		(* split slave state and link state *)
			FOR I_X1 := 1 TO MIN(nEcSlavesRead_X1, GVL.ECAT_MAX_SLAVES_X1) DO
				(* slave state*)
				arrSlaveInfo_X1[I_X1].stState.eEcState 				:= ArrEcSlaveState_X1[I_X1].deviceState AND 16#0F;
				arrSlaveInfo_X1[I_X1].stState.bError 					:= ArrEcSlaveState_X1[I_X1].deviceState.4;
				arrSlaveInfo_X1[I_X1].stState.bInvalidVPRS 			:= ArrEcSlaveState_X1[I_X1].deviceState.5;
				(* link state *)
				arrSlaveInfo_X1[I_X1].stState.bNoCommToSlave 	:= ArrEcSlaveState_X1[I_X1].linkState.0;
				arrSlaveInfo_X1[I_X1].stState.bLinkError 				:= ArrEcSlaveState_X1[I_X1].linkState.1;
				arrSlaveInfo_X1[I_X1].stState.bMissingLink 			:= ArrEcSlaveState_X1[I_X1].linkState.2;
				arrSlaveInfo_X1[I_X1].stState.bUnexpectedLink		:= ArrEcSlaveState_X1[I_X1].linkState.3;
				arrSlaveInfo_X1[I_X1].stState.bPortA 					:= ArrEcSlaveState_X1[I_X1].linkState.4;
				arrSlaveInfo_X1[I_X1].stState.bPortB 					:= ArrEcSlaveState_X1[I_X1].linkState.5;
				arrSlaveInfo_X1[I_X1].stState.bPortC 					:= ArrEcSlaveState_X1[I_X1].linkState.6;
				arrSlaveInfo_X1[I_X1].stState.bPortD 					:= ArrEcSlaveState_X1[I_X1].linkState.7;
				(* DiagData *)
				arrSlaveInfo_X1[I_X1].bDiagData	:= ((ArrEcSlaveState_X1[I_X1].deviceState AND 16#F0) <> 0) OR
					(((ArrEcSlaveState_X1[I_X1].deviceState AND 16#0F) > 0) AND ((ArrEcSlaveState_X1[I_X1].deviceState AND 16#0F) < 8)) OR
					(ArrEcSlaveState_X1[I_X1].linkState <> 0);

				IF arrSlaveInfo_X1[I_X1].bDiagData THEN
					IF (I_X1=0) THEN
						iDiagIndex_X1[0] := 0;
					ELSE
						IF (iDiagIndex_X1[0] = 0) AND NOT arrSlaveInfo_X1[1].bDiagData THEN
							iDiagIndex_X1[0] :=  DINT_TO_UINT(I_X1);
						END_IF
					END_IF
				END_IF


				arrSlaveInfo_X1[I_X1].sName							:=	ArrEcConfSlaveInfo_X1[I_X1].sName;
				arrSlaveInfo_X1[I_X1].sType							:=	ArrEcConfSlaveInfo_X1[I_X1].sType;
				arrSlaveInfo_X1[I_X1].nECAddr						:=	ArrEcConfSlaveInfo_X1[I_X1].nAddr;

				IF arrSlaveInfo_X1[I_X1].stState.bError THEN
					sState_X1	 	:=	'ERR';
				ELSE
					sState_X1		:=	'';
				END_IF

				IF arrSlaveInfo_X1[I_X1].stState.bInvalidVPRS THEN
					sState_X1	 	:=	' VPRS INIT_ERR';
				END_IF

				IF arrSlaveInfo_X1[I_X1].stState.bNoCommToSlave THEN
					sState_X1	 	:=	CONCAT ( sState_X1, ' NO_COMM');
				END_IF

				IF arrSlaveInfo_X1[I_X1].stState.bLinkError THEN
					sState_X1	 	:=	CONCAT ( sState_X1, ' LINK_ERR');
				END_IF

				IF arrSlaveInfo_X1[I_X1].stState.bUnexpectedLink THEN
					sState_X1	 	:=	CONCAT ( sState_X1, ' UNEXP_LINK');
				END_IF

				IF arrSlaveInfo_X1[I_X1].stState.bMissingLink THEN
					sState_X1	 	:=	CONCAT ( sState_X1, ' LINK_MIS ');
				END_IF

				IF arrSlaveInfo_X1[I_X1].stState.bPortA THEN
					sState_X1	 	:=	CONCAT ( sState_X1, 'A ');
				END_IF

				IF arrSlaveInfo_X1[I_X1].stState.bPortB THEN
					sState_X1	 	:=	CONCAT ( sState_X1, 'B ');
				END_IF


				IF arrSlaveInfo_X1[I_X1].stState.bPortC THEN
					sState_X1	 	:=	CONCAT ( sState_X1, 'C ');
				END_IF

				IF arrSlaveInfo_X1[I_X1].stState.bPortD THEN
					sState_X1	 	:=	CONCAT ( sState_X1, 'D ');
				END_IF

				arrSlaveInfo_X1[I_X1].sStateString := sState_X1;
				
				CASE  arrSlaveInfo_X1[I_X1].stState.eEcState	OF 
						
						0:	arrSlaveInfo_X1[I_X1].sEcState	:= 'Úndefined';
						1:	arrSlaveInfo_X1[I_X1].sEcState	:= 'INIT';
						2:	arrSlaveInfo_X1[I_X1].sEcState	:= 'PREOP';
						3:	arrSlaveInfo_X1[I_X1].sEcState	:= 'BOOT';
						4:	arrSlaveInfo_X1[I_X1].sEcState	:= 'SAFEOP';
						8:	arrSlaveInfo_X1[I_X1].sEcState	:= 'OP';
						
				END_CASE
			END_FOR
		END_IF
	END_IF
END_IF

IF bCheckError THEN
		IF N_X1 = 0 THEN
			N_X1 :=1;
		END_IF
		IF arrSlaveInfo_X1[N_X1].sEcState <> 'OP' AND arrSlaveInfo_X1[N_X1].sEcState <> '' THEN
			CASE ErrorState_X1 OF 
				0:
					fbGetSlaveState_X1(sNetId:= sEcMasterNetId_X1,
									   nSlaveAddr:= arrSlaveInfo_X1[N_X1].nECAddr, 
									   bExecute:=TRUE,
									   tTimeout:= DEFAULT_ADS_TIMEOUT,
									   state:=EC_DEVICE_STATE_ERROR);
					ErrorState_X1 := ErrorState_X1+1;
					
				2:
					IF NOT fbGetSlaveState_X1.bBusy AND NOT fbGetSlaveState_X1.bError THEN
						fbGetSlaveState_X1(bExecute:=FALSE);
						ErrorState_X1 := ErrorState_X1+1;
					END_IF
					IF fbGetSlaveState_X1.bBusy AND fbGetSlaveState_X1.bError THEN
						ErrorState_X1 := 100;
					END_IF
				3:
					fbGetSlaveState_X1(sNetId:= sEcMasterNetId_X1,
									   nSlaveAddr:= arrSlaveInfo_X1[N_X1].nECAddr, 
									   bExecute:=TRUE,
									   tTimeout:= DEFAULT_ADS_TIMEOUT,
									   state:=EC_DEVICE_STATE_OP);
					ErrorState_X1 := ErrorState_X1+1;
				4:
					IF NOT fbGetSlaveState_X1.bBusy AND NOT fbGetSlaveState_X1.bError THEN
						fbGetSlaveState_X1(bExecute:=FALSE);
						ErrorState_X1 := ErrorState_X1+1;
					END_IF
					IF fbGetSlaveState_X1.bBusy AND fbGetSlaveState_X1.bError THEN
						ErrorState_X1 := 100;
					END_IF
				5:
					ErrorState_X1 := 0;
					N_X1 := N_X1+1;
			END_CASE;
		ELSE
			N_X1 := N_X1+1;
		END_IF;
		
		IF N_X1 = MIN(nEcSlavesRead_X1, GVL.ECAT_MAX_SLAVES_X1) THEN
			N_X1 := 1;
			bCheckError:=1;
		END_IF
END_IF;

END_PROGRAM

// ---- FB/Cylinder_Block_HOMING.TcPOU
FUNCTION_BLOCK Cylinder_Block_HOMING
VAR_INPUT
	Auto :BOOL;
	Manual :BOOL;
	HOMING_RUNNING:BOOL;
	ErrorActive :BOOL;
	ResetPB :BOOL;
	Sensor1 :BOOL;
	Sensor2 :BOOL;
	ManualPB1 :BOOL;
	ManualPB2 :BOOL;
	AutoCmd1 :BOOL;
	AutoCmd2 :BOOL;
	OperationEnable :BOOL;
	SafeHome :BOOL;
	SafeWork :BOOL;
	Pulse_1Sec :BOOL;
	BlinkingBit :BOOL;
	TimeOut1 :INT;
	TimeOut2 :INT;
	TimeOut3 :INT;
	HOMING_STRT:BOOL;
	HME_DLY:INT;
	HME_DN_NO:INT;
	HME_CYL_2:BOOL;
	HME_CYL_3:BOOL;
END_VAR
VAR_OUTPUT
	Solenoid1 :BOOL;
	Solenoid2 :BOOL;
	AlarmSensor1 :BOOL;
	AlarmSensor2 :BOOL;
	AlarmSolenoid1 :BOOL;
	AlarmSolenoid2 :BOOL;
	AllSignal :BOOL;
	AlarmPresent :BOOL;
	Position1 :BOOL;
	Position2 :BOOL;
	HomeSensorBlink :BOOL;
	WorkSensorBlink :BOOL;
END_VAR
VAR_IN_OUT
	Status :INT;
	HMENG_RESULT: INT;
END_VAR
VAR
	Timer1 :INT;
	Timer2 :INT;
	Timer3 :INT;
	HomingCmd1:BOOL;
	HomePositionErr_1SecPls :Tc2_Standard.R_TRIG;
	WorkPositionErr_1SecPls :Tc2_Standard.R_TRIG;
	BothSensorErr_1SecPls :Tc2_Standard.R_TRIG;
	Temp4 :BOOL;
	AFT_CYL_HME: TON;
END_VAR

Status:=0;
//Cylinder Moving to Home Position by Manual

IF ManualPB1 THEN
	IF NOT Manual THEN Status :=1; 
	ELSIF ManualPB2 THEN Status :=2; 
	ELSIF AllSignal THEN Status :=3;
	ELSIF NOT OperationEnable THEN Status :=9; 
	ELSIF Status =0 AND SafeHome THEN
		Solenoid1 :=1;
		Solenoid2 :=0;
	END_IF 
END_IF


//Cylinder Moving to Work Position by Manual

IF ManualPB2 THEN
	IF NOT Manual THEN Status :=1; 
	ELSIF ManualPB1 THEN Status :=2; 
	ELSIF AllSignal THEN Status :=3;
	ELSIF NOT OperationEnable THEN Status :=9; 
	ELSIF Status =0 AND SafeWork THEN
		Solenoid2 :=1;
		Solenoid1 :=0;
	END_IF 
END_IF


//Cylinder Moving to Home Position by Auto

IF AutoCmd1 THEN
	IF NOT Auto THEN Status :=5; 
	ELSIF AutoCmd2 THEN Status :=6;
	ELSIF ErrorActive THEN Status :=4; 
	ELSIF AllSignal THEN Status :=3;
	ELSIF NOT OperationEnable THEN Status :=9;
	ELSIF Status =0 AND SafeHome THEN
		Solenoid1 :=1;
		Solenoid2 :=0;
	END_IF 
END_IF

//Cylinder Moving to Work Position by Auto

IF AutoCmd2 THEN
	IF NOT Auto THEN Status :=5; 
	ELSIF AutoCmd1 THEN Status :=6;
	ELSIF ErrorActive THEN Status :=4; 
	ELSIF AllSignal THEN Status :=3;
	ELSIF NOT OperationEnable THEN Status :=9;
	ELSIF Status =0 AND SafeWork THEN
		Solenoid2 :=1;
		Solenoid1 :=0;
	END_IF 
END_IF


//Cylinder Moving to Home Position - Homing Cmd ON

IF HomingCmd1 THEN 
	IF AllSignal THEN Status :=3;
	ELSIF NOT OperationEnable THEN Status :=9; 
	ELSIF Status =0 AND SafeHome THEN
		Solenoid1 :=1;
		Solenoid2 :=0;
	END_IF 
END_IF


// While Cylinder Moving Blinking IF Position Reached then Steady Indication

HomeSensorBlink := (Solenoid1 AND NOT Sensor1 AND BlinkingBit) OR Sensor1;
WorkSensorBlink := (Solenoid2 AND NOT Sensor2 AND BlinkingBit) OR Sensor2;


// Position 1 Reached - Cylinder Timer OFF

IF NOT Solenoid1 THEN Timer1 :=0; END_IF


//Timer1 is for Monitoring Cylinder Home Position Time
HomePositionErr_1SecPls(CLK := Pulse_1Sec);

IF Solenoid1 AND NOT Sensor1 AND HomePositionErr_1SecPls.Q THEN 
Timer1 := Timer1 + 1;
ELSE
Timer1	:= 0;	
END_IF


//Generate Alarm for Home Position Sensor & Valve

IF Timer1 >= TimeOut1 AND NOT Sensor1 AND NOT Sensor2 THEN AlarmSensor1 :=1; END_IF
IF Timer1 >= TimeOut1 AND NOT Sensor1 AND Sensor2 THEN AlarmSolenoid1 :=1; END_IF


// Position 2 Reached - Cylinder Timer OFF

IF NOT Solenoid2 THEN Timer2 :=0; END_IF


//Timer2 is for Monitoring Cylinder Work Position Time
WorkPositionErr_1SecPls(CLK := Pulse_1Sec);

IF Solenoid2 AND NOT Sensor2 AND WorkPositionErr_1SecPls.Q THEN 
	Timer2 := Timer2 + 1;
ELSE
	Timer2	:=0;
END_IF


//Generate Alarm for Work Position Sensor & Valve

IF Timer2 >= TimeOut2 AND NOT Sensor2 AND NOT Sensor1 THEN AlarmSensor2 :=1; END_IF
IF Timer2 >= TimeOut2 AND NOT Sensor2 AND Sensor1 THEN AlarmSolenoid2 :=1; END_IF


//Move "0" to Timer3 If anyone Sensor is not Sensing

IF NOT Sensor1 AND NOT Sensor2 THEN Timer3 :=0; END_IF


//Timer3 is for Monitoring Both Sensor ON Error
BothSensorErr_1SecPls (CLK := Pulse_1Sec);

 IF Sensor1 AND Sensor2 AND BothSensorErr_1SecPls.Q THEN
	 Timer3 := Timer3 + 1;
 END_IF
 
 
 //Generate Alarm for Both Sensor ON Error
 
 IF Timer3 >= TimeOut3 THEN AllSignal :=1; END_IF
 
 
 //Reset the Valve when Operation Enable not Present
 
 IF NOT OperationEnable THEN
	 Solenoid1 :=0;
	 Solenoid2 :=0;
 END_IF

 
//Position 1 is Cylinder Home Position || Position 2 is Cylinder Work Position

Position1 := NOT AllSignal AND Sensor1 AND NOT Sensor2;
Position2 := NOT AllSignal AND Sensor2 AND NOT Sensor1; 

// HOMING LOGIC

IF HOMING_RUNNING AND HOMING_STRT AND NOT ErrorActive THEN
	HomingCmd1				:= TRUE;
ELSE
	HomingCmd1				:= FALSE;
END_IF

AFT_CYL_HME(IN:= (HomingCmd1 AND HME_CYL_2 AND HME_CYL_3 AND Sensor1 AND NOT ErrorActive), PT:=INT_TO_TIME(HME_DLY) , Q=> , ET=> );
IF AFT_CYL_HME.Q THEN
	HMENG_RESULT:=HME_DN_NO;
END_IF

// ALARM RESET

IF ResetPB THEN
	
AlarmSensor1 								:= FALSE;
AlarmSensor2            					:= FALSE;
AlarmSolenoid1          					:= FALSE;
AlarmSolenoid2          					:= FALSE;
AllSignal               					:= FALSE;

END_IF


IF AlarmSensor1 OR AlarmSensor2 OR AlarmSolenoid1 OR AlarmSolenoid2 OR AllSignal THEN
		AlarmPresent						:= TRUE;
ELSE
		AlarmPresent						:= FALSE;
END_IF

END_FUNCTION_BLOCK

// ---- FB/Axis/FB_Axis_FESTO.TcPOU
FUNCTION_BLOCK FB_Axis_FESTO
VAR_INPUT
	bAxis1_Ref_Switch 	 : BOOL;//HW-IN
	bInit 				 : BOOL;
	bErrorReset			 : BOOL;//FP Reset Axis Error
	bEnable 			 : BOOL;//Power on
	bMoveVelocity 		 : BOOL;
	bHalt				 : BOOL;//Stop Absolute or Relative movement
	bManualMode			 : BOOL;
	bmove_home			 : BOOL;
	fHomePos 			 : LREAL := 0.0;
	fOverride 			 : LREAL ;//:= 100.0;
	fTargetPosition 	 : LREAL ;//:=  10.0;
	fTargetVelocity 	 : LREAL ; //:= 100.0;
	fAcc				 : LREAL; //:= 100.0;
	fDec				 : LREAL; //:= 100.0;
	Servo_High_Limit	 : LREAL;
	Servo_Low_Limit	 	 : LREAL;
	WARNING_LIMIT		 : LREAL;
	Safe_move_Conditions : BOOL;
	LIMIT_BYPASS		 : BOOL := TRUE;
	TORQUE_APPLIED: LREAL;
END_VAR
VAR_IN_OUT
	Axis 				: AXIS_REF;
	bHome 				: BOOL;
	bSetPosition		: BOOL;//Set Position to HomePos
	bMoveAbsolute 		: BOOL;
	bMoveRelative 		: BOOL;
	bMoveTorque			: BOOL;
    stManualModeAxis  	: stManualModeAxis;
														(*bmove_home			: BOOL;*)
END_VAR

VAR_OUTPUT
	sAxisState			: STRING := '';
	bAxis_ready			: BOOL := 0;
	bAxisInPosition		: BOOL := 0;//In Position or In Target Velocity
	bAxisError			: BOOL := 0;
	bAxisEnabled 		: BOOL := 0;//Power ON
	bAxisHomed			: BOOL := 0;
	bSetPositionDone	: BOOL := 0;
	bHaltDone			: BOOL := 0;
	bSTOPDone			: BOOL := 0;
	bHomeDone			: BOOL := 0;
	bDone				: BOOL := 0;//bMoveAbsolute + bMoveRelative
	bTorqueReached		: BOOL := 0;
	bsafe_to_move		: BOOL;
	baxis_in_home_pos	: BOOL;
	bABS_Pos_done		: BOOL;
	Actual_position		: LREAL;
	Actual_velocity		: LREAL;
	Actual_Torque		: LREAL;
    SERVO_LIMIT_WARNING	: BOOL;	
	
END_VAR
VAR
	temp : LREAL;
	fbAxisReset					: MC_Reset;
	fbAxisPower					: MC_Power;
	fbAxisStop        			: MC_Stop;
	fbAxisHalt        			: MC_Halt;
(*	fbAxisHome					: MC_Home;*)
	fbAxisHome					: Festo_MC_Home;
	fbAxisSetPosition 			: MC_SetPosition;
	fbAxisJog 					: MC_Jog;
	fbAxisMoveAbsolute			: MC_MoveAbsolute;
	fbAxisMoveRelative 			: MC_MoveRelative;
	fbAxisMoveVelocity			: MC_MoveVelocity;
	fbAxisTorqueControl			: MC_TorqueControl;
//Brake Controll
	fbEcCoeSdoRead				: FB_EcCoeSdoRead;
	fbEcCoeSdoWrite				: FB_EcCoeSdoWrite;
	mcReadDriveAddress 			: MC_ReadDriveAddress;
    vendorId   					: BOOL;//Struct HMI Brake open
	bBrakeStateOld 				: BOOL;

//Status Information
	bAxisIsEnabled 				: BOOL;
	bAxisIsHomed 				: BOOL;
	bAxisInError 				: BOOL;
	fActualTorque 				: LREAL;	

//Allgemein
	iSchritt 					: ENUM_Axis;
	bHMFPErrorReset 			: BOOL;
	bFPErrorReset 				: BOOL;
	
	bAxisResetExecute			: BOOL;
	bAxisPowerExecute			: BOOL;
	bAxisStopExecute        	: BOOL;
	bAxisHaltExecute        	: BOOL;
	bAxisHomeExecute			: BOOL;
	bAxisSetPositionExecute 	: BOOL;
	bAxisMoveAbsoluteExecute	: BOOL;
	bAxisMoveRelativeExecute 	: BOOL;
	bAxisMoveVelocityExecute	: BOOL;
	bAxisJogExecutePos 			: BOOL;
	bAxisJogExecuteNeg 			: BOOL;
	bAxisMoveTorqueExecute		: BOOL;
	fHMTargetPosition			: LREAL;
	fHMTargetVelocity			: LREAL;
	
	bFPManualReset				: BOOL;
	bHMFPManualReset			: BOOL;
	
	homeMode					: MC_HomingMode;
	FB_SoEReset					: FB_SoEReset;
	bHardwareReset				: BOOL;

	st_Trq_options 				: St_TorqueControlOptions;
	//temp						: BOOL;
	moving_home					: INT;
	bABS_done					: BOOL;
	busy: BOOL;
	act: BOOL;
	id: UDINT;
	AXIS_REF_TEMP: BOOL;
	
	LEG_LIMIT: BOOL;
	POS_LIMIT: BOOL;
	AUTO_TARGET_POSITION: LREAL;
	MANUAL_TARGET_POSITION: LREAL;
	ABS_BUSY: R_TRIG;
END_VAR
VAR_TEMP
 	//tmpVelocityDirection		: MC_Direction;
	tmpStManualModeAxis	  		: stManualModeAxis;
	btmpFPBrake					: BOOL;
//	tmpVelocityDirection        : MC_Direction;
END_VAR


//Init
bHaltDone := FALSE;
bSTOPDone := FALSE;

//Read Axis Status	
	bAxisIsEnabled := axis.NcToPlc.StateDWord.0;
	bAxisIsHomed := axis.NcToPlc.StateDWord.1 OR NOT AXIS_REF_TEMP;
	bAxisInError := axis.NcToPlc.StateDWord.31;
	fActualTorque := axis.NcToPlc.ActTorque;
    Axis.ReadStatus(); // PHU: fill its own status bits.
//FP Error Reset
	bFPErrorReset := bErrorReset (*AND NOT bHMFPErrorReset*);
	bHMFPErrorReset := bErrorReset;
	
	bFPManualReset:= stManualModeAxis.reset AND NOT bHMFPManualReset;
	bHMFPManualReset:= stManualModeAxis.reset;
	
// Manual Mode
IF bManualMode THEN
	
	stManualModeAxis.stationModeAutoManual:= FALSE;	
	IF 	stManualModeAxis.jogPos THEN
		tmpStManualModeAxis.jogPos := TRUE;
	ELSE
		tmpStManualModeAxis.jogPos := FALSE;		
	END_IF
	IF 	stManualModeAxis.jogNeg THEN
		tmpStManualModeAxis.jogNeg := TRUE;
	ELSE
		tmpStManualModeAxis.jogNeg := FALSE;		
	END_IF
		
ELSE
	stManualModeAxis.jogPos := FALSE;
	stManualModeAxis.jogNeg := FALSE;
	stManualModeAxis.reset := FALSE;
	StManualModeAxis.openBrake:= FALSE;
	stManualModeAxis.homing:= FALSE;
	stManualModeAxis.moveAbsolute:= FALSE;
	stManualModeAxis.moveRelative:= FALSE;
	stManualModeAxis.moveVelocity:= FALSE;
	
	tmpStManualModeAxis.jogPos := FALSE;		
	tmpStManualModeAxis.jogNeg := FALSE;	
	
	
	
	stManualModeAxis.stationModeAutoManual:= TRUE;

END_IF


//###################################################################################
//###################################################################################	
	
//###################################################################################
//###################################################################################

	CASE iSchritt OF 
		
	ENUM_Axis.Init 			://init all MC
								bAxisResetExecute				:= FALSE;
								bAxisPowerExecute				:= FALSE;
								bAxisStopExecute        		:= FALSE;
								bAxisHaltExecute        		:= FALSE;
								bAxisHomeExecute				:= FALSE;
								bAxisSetPositionExecute 		:= FALSE;
								bAxisJogExecutePos 				:= FALSE;
								bAxisJogExecuteNeg 				:= FALSE;
								bAxisMoveAbsoluteExecute		:= FALSE;
								bAxisMoveRelativeExecute 		:= FALSE;
								bAxisMoveVelocityExecute		:= FALSE;
								
								iSchritt := ENUM_Axis.PowerOFF;
								

	ENUM_Axis.PowerOFF		: 	//Power off
								bAxisPowerExecute		:= FALSE;
								IF bInit THEN
									iSchritt := ENUM_Axis.Init;
								ELSIF bAxisInError THEN
									iSchritt := ENUM_Axis.Error;
								ELSIF bEnable THEN
									iSchritt := ENUM_Axis.PowerON;
								END_IF
								
	ENUM_Axis.Error			:	//Error
								bAxisPowerExecute			  := FALSE;
								bMoveAbsolute				  := FALSE;
								bMoveRelative			   	  := FALSE;
								stManualModeAxis.moveAbsolute := FALSE;
								stManualModeAxis.moveRelative := FALSE;
								IF bInit THEN
									iSchritt := ENUM_Axis.Init;
								ELSIF bFPErrorReset OR bFPManualReset THEN
									iSchritt := ENUM_Axis.Reset;
								END_IF
	ENUM_Axis.Reset			: //Error Reset
								IF NOT fbAxisReset.Busy THEN
									bAxisResetExecute 		:= TRUE;
									bHardwareReset			:= axis.NcToPlc.StateDWord.28;
								END_IF;
								IF bInit THEN
									bAxisResetExecute 		:= FALSE;
									iSchritt := ENUM_Axis.Init;
								ELSIF fbAxisReset.Error (*OR bAxisInError *)THEN
									bAxisResetExecute 	:= FALSE;
									iSchritt := ENUM_Axis.Error;
								ELSIF fbAxisReset.Done AND NOT bAxisInError THEN
									bAxisResetExecute 	:= FALSE;
									IF  bAxisInError THEN
										iSchritt := ENUM_Axis.Error;
									ELSE
										iSchritt := ENUM_Axis.PowerOFF;
									END_IF
								END_IF

	ENUM_Axis.PowerON		:	//Enable - Power on
								bAxisPowerExecute := TRUE;
								IF bInit THEN
									bAxisPowerExecute 	:= FALSE;
									iSchritt := ENUM_Axis.Init;
								ELSIF NOT benable THEN
									iSchritt:= enum_axis.PowerOFF;
								ELSIF fbAxisPower.Error OR bAxisInError THEN
									bAxisPowerExecute 	:= FALSE;
									iSchritt := ENUM_Axis.Error;
								ELSIF fbAxisPower.Status THEN
									iSchritt := ENUM_Axis.Ready;
								END_IF
	ENUM_Axis.Stop			://Axis Stop
								bAxisStopExecute := TRUE;
								IF bInit THEN
									bAxisStopExecute 	:= FALSE;
									iSchritt := ENUM_Axis.Init;
								ELSIF NOT benable THEN
									bAxisStopExecute 	:= FALSE;
									iSchritt:= enum_axis.PowerOFF;	
								ELSIF fbAxisStop.Error OR bAxisInError THEN
									bAxisStopExecute := FALSE;
									iSchritt := ENUM_Axis.Error;
								ELSIF fbAxisStop.Done THEN
									bSTOPDone	:= TRUE;
									bAxisStopExecute 	:= FALSE;
									iSchritt := ENUM_Axis.PowerOFF;
								END_IF
	ENUM_Axis.Halt			://Axis Halt
								bAxisHaltExecute := TRUE;
								IF bInit THEN
									bAxisHaltExecute 	:= FALSE;
									iSchritt := ENUM_Axis.Init;
								ELSIF NOT benable THEN
									bAxisHaltExecute 	:= FALSE;
									iSchritt:= enum_axis.PowerOFF;	
								ELSIF bAxisInError THEN
									bAxisHaltExecute := FALSE;
									iSchritt := ENUM_Axis.Error;
								ELSIF fbAxisHalt.Error (*OR bAxisInError *)THEN
									bAxisHaltExecute := FALSE;
									iSchritt := ENUM_Axis.Stop;
								ELSIF fbAxisHalt.Done THEN
									bHaltDone := TRUE;
									bAxisHaltExecute := FALSE;
									iSchritt := ENUM_Axis.Ready;
								END_IF
	ENUM_Axis.Ready			: 	//Wait for command
								bAxisInPosition := FALSE;
								//bHomeDone := FALSE;
								bSetPositionDone := FALSE;
								IF bInit THEN
									iSchritt := ENUM_Axis.Init;
								ELSIF NOT benable THEN
									iSchritt:= enum_axis.PowerOFF;		
								ELSIF bAxisInError THEN
									iSchritt := ENUM_Axis.Error;
								ELSE
									IF bHome OR stManualModeAxis.homing THEN
										iSchritt := ENUM_Axis.Homing;
									ELSIF bSetPosition THEN
											iSchritt := ENUM_Axis.SetPosition;
									ELSIF bAxisIsHomed THEN
										IF tmpStManualModeAxis.jogPos THEN
											iSchritt := ENUM_Axis.JogPos;
										ELSIF tmpStManualModeAxis.jogNeg THEN
											iSchritt := ENUM_Axis.JogNeg;
										ELSIF bMoveAbsolute OR stManualModeAxis.moveAbsolute  THEN
											iSchritt := ENUM_Axis.MoveAbsolute;
										ELSIF bMoveRelative OR stManualModeAxis.moveRelative THEN
											iSchritt := ENUM_Axis.MoveRelative;
										ELSIF bMoveVelocity OR stManualModeAxis.moveVelocity THEN
											iSchritt := ENUM_Axis.MoveVelocity;
										ELSIF bMoveTorque OR stManualModeAxis.moveTorque THEN
											iSchritt := ENUM_Axis.MoveTorque;
										END_IF
									END_IF	
								END_IF							
	ENUM_Axis.Homing		://Homing
								IF NOT fbAxisHome.Busy THEN
									bAxisHomeExecute := TRUE;
									bHomeDone		:= FALSE;
								END_IF;
								IF bInit THEN
									bAxisHomeExecute 	:= FALSE;
									iSchritt := ENUM_Axis.Init;
								ELSIF NOT benable THEN
									bAxisHomeExecute:= FALSE;
									iSchritt:= enum_axis.PowerOFF;	
								ELSIF fbAxisHome.Error OR bAxisInError THEN
									bAxisHomeExecute:= FALSE;
									iSchritt := ENUM_Axis.Error;
								ELSIF fbAxisHome.Done THEN
									bHomeDone	:= TRUE;
									bHome := FALSE;
									stManualModeAxis.homing:= FALSE;
									bAxisHomeExecute:= FALSE;
									iSchritt := ENUM_Axis.Ready;
								END_IF
	
	ENUM_Axis.SetPosition	://Enable - Power on
								IF NOT fbAxisSetPosition.Busy THEN
									bAxisSetPositionExecute := TRUE;
								END_IF;
								IF bInit THEN
									bAxisSetPositionExecute 	:= FALSE;
									iSchritt := ENUM_Axis.Init;
								ELSIF NOT benable THEN
									bAxisSetPositionExecute 	:= FALSE;
									iSchritt:= enum_axis.PowerOFF;		
								ELSIF fbAxisSetPosition.Error OR bAxisInError THEN
									bAxisSetPositionExecute 	:= FALSE;
									iSchritt := ENUM_Axis.Error;
								ELSIF fbAxisSetPosition.Done THEN
									bAxisSetPositionExecute 	:= FALSE;
									bSetPositionDone := TRUE;
									bSetPosition := FALSE;
									iSchritt := ENUM_Axis.Ready;
								END_IF

	ENUM_Axis.JogPos		://Jog positive direction
								IF NOT fbAxisJog.Busy THEN
									bAxisJogExecutePos 		:= TRUE;
								END_IF;
								
								IF bInit THEN
									bAxisJogExecutePos 	:= FALSE;
									iSchritt := ENUM_Axis.Init;
								ELSIF NOT benable THEN
									bAxisJogExecutePos 	:= FALSE;
									iSchritt:= enum_axis.PowerOFF;			
								ELSIF fbAxisJog.Error OR bAxisInError THEN
									bAxisJogExecutePos 		:= FALSE;
									iSchritt := ENUM_Axis.Error;
								ELSIF NOT tmpStManualModeAxis.jogPos THEN
									bAxisJogExecutePos 		:= FALSE;
									iSchritt := ENUM_Axis.Ready;
								END_IF;
	ENUM_Axis.JogNeg		://Jog negative direction
								IF NOT fbAxisJog.Busy THEN
									bAxisJogExecuteNeg 		:= TRUE;
								END_IF;
								
								IF bInit THEN
									bAxisJogExecuteNeg 	:= FALSE;
									iSchritt := ENUM_Axis.Init;
								ELSIF NOT benable THEN
									bAxisJogExecuteNeg 	:= FALSE;
									iSchritt:= enum_axis.PowerOFF;		
								ELSIF fbAxisJog.Error OR bAxisInError THEN
									bAxisJogExecuteNeg 		:= FALSE;
									iSchritt := ENUM_Axis.Error;
								ELSIF NOT tmpStManualModeAxis.jogNeg THEN
									bAxisJogExecuteNeg 		:= FALSE;
									iSchritt := ENUM_Axis.Ready;
								END_IF;
	ENUM_Axis.MoveAbsolute	://MoveAbsolute
								IF NOT fbAxisMoveAbsolute.Busy THEN
									bAxisMoveAbsoluteExecute := TRUE;
								END_IF;
								IF bInit THEN
									bAxisMoveAbsoluteExecute 	:= FALSE;
									iSchritt := ENUM_Axis.Init;
								ELSIF NOT benable THEN
									bAxisMoveAbsoluteExecute 	:= FALSE;
									iSchritt:= enum_axis.PowerOFF;		
								ELSIF fbAxisMoveAbsolute.Error OR bAxisInError THEN
									bAxisMoveAbsoluteExecute :=FALSE;
									iSchritt := ENUM_Axis.Error;
								ELSIF bHalt THEN
									bMoveAbsolute :=FALSE;
									stManualModeAxis.moveAbsolute:= FALSE;
									bAxisMoveAbsoluteExecute :=FALSE;
									iSchritt := ENUM_Axis.Halt;
								ELSIF fbAxisMoveAbsolute.Done THEN
								//ELSIF fbAxisMoveAbsolute.Done AND NOT bMoveAbsolute THEN
									bMoveAbsolute :=FALSE;
									stManualModeAxis.moveAbsolute:= FALSE;
									bAxisInPosition := TRUE;
									bAxisMoveAbsoluteExecute :=FALSE;
									iSchritt := ENUM_Axis.Ready;
								END_IF;
	ENUM_Axis.MoveRelative	://MoveRelative
								IF NOT fbAxisMoveRelative.Busy THEN
									bAxisMoveRelativeExecute := TRUE;
								END_IF;
								IF bInit THEN
									bAxisMoveRelativeExecute 	:= FALSE;
									iSchritt := ENUM_Axis.Init;
								ELSIF NOT benable THEN
									bAxisMoveRelativeExecute 	:= FALSE;
									iSchritt:= enum_axis.PowerOFF;		
								ELSIF fbAxisMoveRelative.Error OR bAxisInError THEN
									bAxisMoveRelativeExecute :=FALSE;
									iSchritt := ENUM_Axis.Error;
								ELSIF bHalt THEN
									bMoveRelative :=FALSE;
									stManualModeAxis.moveRelative:= FALSE;
									bAxisMoveRelativeExecute :=FALSE;
									iSchritt := ENUM_Axis.Halt;
								ELSIF fbAxisMoveRelative.Done THEN
									bMoveRelative :=FALSE;
									stManualModeAxis.moveRelative:= FALSE;
									bAxisInPosition := TRUE;
									bAxisMoveRelativeExecute :=FALSE;
									iSchritt := ENUM_Axis.Ready;
								END_IF;
	ENUM_Axis.MoveVelocity	://MoveVelocity
								IF NOT fbAxisMoveVelocity.Busy THEN
									bAxisMoveVelocityExecute := TRUE;				
								END_IF;
								
								bAxisInPosition := fbAxisMoveVelocity.InVelocity;
								IF bInit THEN
									bAxisMoveVelocityExecute 	:= FALSE;
									bAxisInPosition := FALSE;
									iSchritt := ENUM_Axis.Init;
								ELSIF NOT benable THEN
									bAxisMoveVelocityExecute 	:= FALSE;
									iSchritt:= enum_axis.PowerOFF;		
								ELSIF fbAxisMoveVelocity.Error OR bAxisInError THEN
									bAxisInPosition := FALSE;
									bAxisMoveVelocityExecute :=FALSE;
									iSchritt := ENUM_Axis.Error;
								ELSIF NOT bMoveVelocity AND NOT stManualModeAxis.moveVelocity THEN
									bAxisInPosition := FALSE;
									bAxisMoveVelocityExecute :=FALSE;
									iSchritt := ENUM_Axis.Halt;
								END_IF;
								
	ENUM_Axis.MoveTorque  :		IF NOT fbAxisTorqueControl.Busy THEN
									bAxisMoveTorqueExecute := TRUE;
								END_IF;
								IF bInit THEN
									bAxisMoveTorqueExecute 	:= FALSE;
									iSchritt := ENUM_Axis.Init;
								ELSIF NOT benable THEN
									bAxisMoveTorqueExecute 	:= FALSE;
									iSchritt:= enum_axis.PowerOFF;		
								ELSIF fbAxisTorqueControl.Error OR bAxisInError THEN
									bAxisMoveTorqueExecute :=FALSE;
									iSchritt := ENUM_Axis.Error;
								ELSIF bHalt THEN
									bMoveTorque	 :=FALSE;
									stManualModeAxis.moveTorque:= FALSE;
									bAxisMoveTorqueExecute :=FALSE;
									iSchritt := ENUM_Axis.Halt;
								ELSIF fbAxisTorqueControl.InTorque THEN
								//ELSIF fbAxisMoveAbsolute.Done AND NOT bMoveAbsolute THEN
									bMoveTorque :=FALSE;
									stManualModeAxis.moveTorque:= FALSE;
									bAxisInPosition := TRUE;
									bAxisMoveTorqueExecute :=FALSE;
									iSchritt := ENUM_Axis.Ready;
								END_IF;					

	END_CASE;
	
	
	stManualModeAxis.axisState:= TO_STRING(iSchritt);
//###################################################################################
//###################################################################################
//###################################################################################
//###################################################################################



fbAxisReset(
	Axis:= Axis, 
	Execute:= bAxisResetExecute , 
	Done=> , 
	Busy=> , 
	Error=> , 
	ErrorID=> );
	
fbAxisPower(
	Axis:= Axis, 
	Enable:= bAxisPowerExecute, 
	Enable_Positive:= bAxisPowerExecute, 
	Enable_Negative:= bAxisPowerExecute, 
	Override:= fOverride, 
	//BufferMode:= , 
	//Options:= , 
	Status=> , 
	Busy=> , 
	Active=> , 
	Error=> , 
	ErrorID=> );
	
fbAxisStop(
	Axis:= Axis, 
	Execute:= bAxisStopExecute, 
	Deceleration:= fDec, 
	Jerk:= 0, 
	//Options:= , 
	Done=> , 
	Busy=> , 
	Active=> , 
	CommandAborted=> , 
	Error=> , 
	ErrorID=> );
	
fbAxisHalt(
	Axis:= Axis, 
	Execute:= bAxisHaltExecute, 
	Deceleration:= fDec, 
	Jerk:= 0, 
	//BufferMode:= , 
	//Options:= , 
	Done=> , 
	Busy=> , 
	Active=>, 
	CommandAborted=> , 
	Error=> , 
	ErrorID=> );

//Homingmode
IF bAxisHomeExecute THEN
	//HomeMode := MC_DefaultHoming;
	HomeMode := MC_Direct;
ELSIF bAxisSetPositionExecute THEN
	//HomeMode := MC_ForceCalibration;
		HomeMode := MC_Direct;
END_IF;


IF bManualMode THEN
	fHMTargetPosition:= MANUAL_TARGET_POSITION;
	fHMTargetVelocity:= stManualModeAxis.targetVelocity;
ELSE
	fHMTargetPosition:=AUTO_TARGET_POSITION;
	fHMTargetVelocity:=fTargetVelocity;
END_IF


(*fbAxisHome(
	Axis:= Axis, 
	Execute:= bAxisHomeExecute OR bAxisSetPositionExecute , 
	Position:= fHomePos, 
	HomingMode:= HomeMode, //MC_DefaultHoming,//, MC_Block
	//BufferMode:= , 
	Options:= , 
	bCalibrationCam:= bAxis1_Ref_Switch, 
	Done=> , 
	Busy=> , 
	Active=> , 
	CommandAborted=> , 
	Error=> , 
	ErrorID=> );*)

fbAxisHome(
	Axis:= Axis, 
	Execute:= bAxisHomeExecute OR bAxisSetPositionExecute , 
	TimeoutTimeHomingRun:= T#1M, 
	Done=> , 
	Busy=> , 
	Error=> , 
	ErrorID=> , 
	ErrorString=> );	
	
fbAxisSetPosition(
	Axis:= Axis, 
	Execute:= bAxisSetPositionExecute, 
	Position:= fHomePos, 
	Mode:= FALSE, (* RELATIVE=True, ABSOLUTE=False (Default) *)
	//Options:= , 
	Done=> , 
	Busy=> , 
	Error=> , 
	ErrorID=> );

fbAxisJog(
	Axis:= Axis, 
	JogForward:=bAxisJogExecutePos AND (POS_LIMIT OR LIMIT_BYPASS),
	JogBackwards:= bAxisJogExecuteNeg AND (LEG_LIMIT OR LIMIT_BYPASS),
	//Mode:= MC_JOGMODE_STANDARD_SLOW, //MC_JOGMODE_STANDARD_SLOW, //MC_JOGMODE_STANDARD_FAST, //MC_JOGMODE_CONTINOUS, //MC_JOGMODE_INCHING, //MC_JOGMODE_INCHING_MODULO
	//Position:= 0, 
	Velocity:= stManualModeAxis.targetVelocity, 
	Acceleration:= fAcc, 
	Deceleration:= fDec, 
	Jerk:= 0, 
	Done=> , 
	Busy=> , 
	Active=> , 
	CommandAborted=> , 
	Error=> , 
	ErrorID=> );
	
fbAxisMoveAbsolute(
	Axis:= Axis, 
	Execute:= bAxisMoveAbsoluteExecute, 
	Position:= fHMTargetPosition,
	Velocity:= ABS(fHMTargetVelocity),
	Acceleration:= fAcc,
	Deceleration:= fDec,
	Jerk:= 0, 
	//BufferMode:= , 
	//Options:= , 
	Done=> , 
	Busy=> , 
	Active=> (bABS_done) , 
	CommandAborted=> , 
	Error=> , 
	ErrorID=> );

	ABS_BUSY(CLK:= bABS_done, Q=> );
	IF ABS_BUSY.Q THEN
	bABS_Pos_done			:= FALSE;	
	END_IF
	IF fbAxisMoveAbsolute.Done THEN
	bABS_Pos_done			:= TRUE;	
	END_IF
	
	
	
fbAxisMoveRelative(
	Axis:= Axis, 
	Execute:= bAxisMoveRelativeExecute, 
	Distance:= fHMTargetPosition, 
	Velocity:= fHMTargetVelocity, 
	Acceleration:= fAcc, 
	Deceleration:= fDec, 
	Jerk:= 0, 
	//BufferMode:= , 
	//Options:= , 
	Done=> , 
	Busy=> , 
	Active=> , 
	CommandAborted=> , 
	Error=> , 
	ErrorID=> );

IF 	fHMTargetVelocity >= 0 THEN  // fHMTargetVelocity>= 0
	fbAxisMoveVelocity.Direction:= MC_Positive_Direction;
ELSE
	fbAxisMoveVelocity.Direction:= MC_Negative_Direction;
END_IF
	
fbAxisMoveVelocity(
	Axis:= Axis, 
	Execute:= bAxisMoveVelocityExecute, 
	Velocity:=ABS(fHMTargetVelocity), 
	Acceleration:= fAcc, 
	Deceleration:= fDec, 
	Jerk:= 0, 
	Direction:= ,//MC_Negative_Direction ,//OR MC_Positive_Direction, //tmpVelocityDirection,//MC_Undefined_Direction, //MC_Shortest_Way, //MC_Positive_Direction, //MC_Negative_Direction,
	//BufferMode:= , 
	//Options:= , 
	InVelocity=> , 
	Busy=> , 
	Active=> , 
	CommandAborted=> , 
	Error=> , 
	ErrorID=> );
	
//Brake controll
vendorId	:= StManualModeAxis.openBrake;	
btmpFPBrake :=  bBrakeStateOld <> vendorId;
bBrakeStateOld := vendorId;

mcReadDriveAddress(
	Axis:= Axis, 
	Execute:= btmpFPBrake, 
	Done=> , 
	Busy=> , 
	Error=> , 
	ErrorID=> , 
	DriveAddress=> Axis.DriveAddress);

	st_Trq_options.EnableManualTorqueStartValue :=TRUE;
	st_Trq_options.ManualTorqueStartValue:= 0.5;
	bTorqueReached:=fbAxisTorqueControl.InTorque;
	
fbAxisTorqueControl	(
	Axis:= Axis , 
	Execute:=bAxisMoveTorqueExecute , 
	Relative:= , 
	Torque:= TORQUE_APPLIED, 
	TorqueRamp:= 50, 
	VelocityLimitHigh:= 500, 
	VelocityLimitLow:= -500, 
	BufferMode:= , 
	Options:= ,//st_Trq_options , 
	InTorque=> , 
	Busy=> busy, 
	Active=> , 
	CommandAborted=> , 
	Error=> act, 
	ErrorId=> id );

//	fbEcCoeSdoRead(
//	sNetId:= Axis.DriveAddress.NetID,
//	nSlaveAddr:= Axis.DriveAddress.SlaveAddress,
//	nSubIndex:= 16#1, 
//	nIndex:= 16#8012, 
//	pDstBuf:= ADR(bBrakeStateOld), 
//	cbBufLen:= SIZEOF(bBrakeStateOld), 
//	bExecute:= mcReadDriveAddress.done, 
//	tTimeout:= , 
//	bBusy=> , 
//	bError=> , 
//	nErrId=> , 
//	cbRead=> );

fbEcCoeSdoWrite(
	sNetId:= Axis.DriveAddress.NetID,
	nSlaveAddr:= Axis.DriveAddress.SlaveAddress, 
	nSubIndex:= 16#1, 
	nIndex:= 16#8012, 
	pSrcBuf:= ADR(bBrakeStateOld), 
	cbBufLen:= SIZEOF(bBrakeStateOld), 
	bExecute:= mcReadDriveAddress.done, 
	tTimeout:= , 
	bBusy=> , 
	bError=> , 
	nErrId=> );
	
			IF bHardwareReset THEN
				FB_SoEReset(
				Axis:= Axis,	
				Execute:= TRUE,
				);
				IF NOT FB_SoEReset.Busy THEN
					FB_SoEReset(
					Axis:= Axis,	
					Execute:= FALSE,
					);
					bHardwareReset:= FALSE;
				END_IF	
			END_IF		

stManualModeAxis.actualPosition:=axis.NcToPlc.ActPos;
stManualModeAxis.actualVelocity:=axis.NcToPlc.ActVelo;
Actual_Torque:=fActualTorque;
//###################################################################################
//###################################################################################

//Output Signals
	sAxisState := TO_STRING(iSchritt);
	bAxisHomed := bAxisIsHomed;
	bAxisError := bAxisInError OR iSchritt = ENUM_Axis.Error;
	bAxis_ready := (iSchritt = ENUM_Axis.Ready);
	
IF In_range(stManualModeAxis.actualPosition,0,1) THEN
	baxis_in_home_pos:=TRUE;
ELSE
	baxis_in_home_pos:=FALSE;		
END_IF	
	
IF Safe_move_Conditions THEN
	bsafe_to_move:=TRUE;
	fOverride := 100;
ELSE
	bsafe_to_move:=FALSE;
	fOverride := 0;
END_IF	

(*IF bmove_home THEN
	CASE moving_home OF
		0:IF bmove_home AND NOT bMoveAbsolute AND NOT baxis_in_home_pos THEN
            fTargetPosition:=0;
		    moving_home:=1;	
		  ELSIF baxis_in_home_pos THEN
			bmove_home:=FALSE;
			moving_home:=0;		
		  END_IF
	   
		1: bMoveAbsolute:=TRUE; 
		   moving_home:=2;  
		
		2:  IF In_range(stManualModeAxis.actualPosition,0,1) OR bDone THEN
			 bMoveAbsolute:=FALSE;
			// moving_home:=0;
			 bmove_home:=FALSE;
		    END_IF		
	END_CASE
ELSE
	moving_home:=0;
END_IF*)

Actual_position:=stManualModeAxis.actualPosition;
Actual_velocity:=stManualModeAxis.actualVelocity;


bAxisEnabled:= NOT bAxisError AND fbAxisPower.Status;

//############################################################


IF NOT LIMIT_BYPASS THEN

IF (stManualModeAxis.actualPosition>=Servo_Low_Limit) THEN
	LEG_LIMIT			:= TRUE;
ELSE	
	LEG_LIMIT			:= FALSE;
END_IF;

IF stManualModeAxis.actualPosition<=Servo_High_Limit THEN
	POS_LIMIT			:= TRUE;	
ELSE
	POS_LIMIT			:= FALSE;
END_IF
 
IF (fTargetPosition<=Servo_High_Limit) AND (fTargetPosition>=Servo_Low_Limit) THEN
	AUTO_TARGET_POSITION:=fTargetPosition;
ELSIF (fTargetPosition>=Servo_High_Limit)THEN
	AUTO_TARGET_POSITION:=Servo_High_Limit;
ELSIF (fTargetPosition<=Servo_Low_Limit) AND (fTargetPosition<=Servo_High_Limit) THEN
	AUTO_TARGET_POSITION:=Servo_Low_Limit;	
END_IF

IF (stManualModeAxis.targetPositon<=Servo_High_Limit) AND (stManualModeAxis.targetPositon>=Servo_Low_Limit) THEN
	MANUAL_TARGET_POSITION:=stManualModeAxis.targetPositon;
ELSIF (stManualModeAxis.targetPositon>=Servo_High_Limit)THEN
	MANUAL_TARGET_POSITION:=Servo_High_Limit;
ELSIF (stManualModeAxis.targetPositon<=Servo_Low_Limit) AND (stManualModeAxis.targetPositon<=Servo_High_Limit) THEN
	MANUAL_TARGET_POSITION:=Servo_Low_Limit;	
END_IF

IF (stManualModeAxis.actualPosition-WARNING_LIMIT)<=Servo_Low_Limit AND (stManualModeAxis.actualPosition+WARNING_LIMIT)<=Servo_High_Limit THEN
	SERVO_LIMIT_WARNING	:= TRUE;
ELSE
	SERVO_LIMIT_WARNING	:= FALSE;	
END_IF

ELSE	
	AUTO_TARGET_POSITION			:=fTargetPosition;
	MANUAL_TARGET_POSITION			:=stManualModeAxis.targetPositon;
END_IF

END_FUNCTION_BLOCK

// ---- FB/Cylinder_Block.TcPOU
FUNCTION_BLOCK Cylinder_Block
VAR_INPUT
	Auto :BOOL;
	Manual :BOOL;
	ErrorActive :BOOL;
	ResetPB :BOOL;
	Sensor1 :BOOL;
	Sensor2 :BOOL;
	ManualPB1 :BOOL;
	ManualPB2 :BOOL;
	AutoCmd1 :BOOL;
	AutoCmd2 :BOOL;
	OperationEnable :BOOL;
	SafeHome :BOOL;
	SafeWork :BOOL;
	HomingCmd1 :BOOL;
	Pulse_1Sec :BOOL;
	BlinkingBit :BOOL;
	TimeOut1 :INT;
	TimeOut2 :INT;
	TimeOut3 :INT;
END_VAR
VAR_OUTPUT
	Solenoid1 :BOOL;
	Solenoid2 :BOOL;
	AlarmSensor1 :BOOL;
	AlarmSensor2 :BOOL;
	AlarmSolenoid1 :BOOL;
	AlarmSolenoid2 :BOOL;
	AllSignal :BOOL;
	AlarmPresent :BOOL;
	Position1 :BOOL;
	Position2 :BOOL;
	HomeSensorBlink :BOOL;
	WorkSensorBlink :BOOL;
END_VAR
VAR_IN_OUT
	Status :INT;
END_VAR
VAR
	Timer1 :INT;
	Timer2 :INT;
	Timer3 :INT;
	HomePositionErr_1SecPls :Tc2_Standard.R_TRIG;
	WorkPositionErr_1SecPls :Tc2_Standard.R_TRIG;
	BothSensorErr_1SecPls :Tc2_Standard.R_TRIG;
	Temp4 :BOOL;
END_VAR

Status:=0;

//Cylinder Moving to Home Position by Manual

IF ManualPB1 THEN
	IF NOT Manual THEN Status :=1; 
	ELSIF ManualPB2 THEN Status :=2; 
	ELSIF AllSignal THEN Status :=3;
	ELSIF NOT OperationEnable THEN Status :=9; 
	ELSIF Status =0 AND SafeHome THEN
		Solenoid1 :=1;
		Solenoid2 :=0;
	END_IF 
END_IF


//Cylinder Moving to Work Position by Manual

IF ManualPB2 THEN
	IF NOT Manual THEN Status :=1; 
	ELSIF ManualPB1 THEN Status :=2; 
	ELSIF AllSignal THEN Status :=3;
	ELSIF NOT OperationEnable THEN Status :=9; 
	ELSIF Status =0 AND SafeWork THEN
		Solenoid2 :=1;
		Solenoid1 :=0;
	END_IF 
END_IF


//Cylinder Moving to Home Position by Auto

IF AutoCmd1 THEN
	IF NOT Auto THEN Status :=5; 
	ELSIF AutoCmd2 THEN Status :=6;
	ELSIF ErrorActive THEN Status :=4; 
	ELSIF AllSignal THEN Status :=3;
	ELSIF NOT OperationEnable THEN Status :=9; 
	ELSIF Status =0 AND SafeHome THEN
		Solenoid1 :=1;
		Solenoid2 :=0;
	END_IF 
END_IF


//Cylinder Moving to Work Position by Auto

IF AutoCmd2 THEN
	IF NOT Auto THEN Status :=5; 
	ELSIF AutoCmd1 THEN Status :=6;
	ELSIF ErrorActive THEN Status :=4; 
	ELSIF AllSignal THEN Status :=3;
	ELSIF NOT OperationEnable THEN Status :=9; 
	ELSIF Status =0 AND SafeWork THEN
		Solenoid2 :=1;
		Solenoid1 :=0;
	END_IF 
END_IF


//Cylinder Moving to Home Position - Homing Cmd ON

IF HomingCmd1 THEN 
	IF AllSignal THEN Status :=3;
	ELSIF NOT OperationEnable THEN Status :=9; 
	ELSIF Status =0 AND SafeHome THEN
		Solenoid1 :=1;
		Solenoid2 :=0;
	END_IF 
END_IF


// While Cylinder Moving Blinking IF Position Reached then Steady Indication

HomeSensorBlink := (Solenoid1 AND NOT Sensor1 AND BlinkingBit) OR Sensor1;
WorkSensorBlink := (Solenoid2 AND NOT Sensor2 AND BlinkingBit) OR Sensor2;


// Position 1 Reached - Cylinder Timer OFF

IF NOT Solenoid1 THEN Timer1 :=0; END_IF


//Timer1 is for Monitoring Cylinder Home Position Time
HomePositionErr_1SecPls(CLK := Pulse_1Sec);

IF Solenoid1 AND NOT Sensor1 AND HomePositionErr_1SecPls.Q THEN 
Timer1 := Timer1 + 1;
ELSE
Timer1:= 0;	
END_IF


//Generate Alarm for Home Position Sensor & Valve

IF Timer1 >= TimeOut1 AND NOT Sensor1 AND NOT Sensor2 THEN AlarmSensor1 :=1; END_IF
IF Timer1 >= TimeOut1 AND NOT Sensor1 AND Sensor2 THEN AlarmSolenoid1 :=1; END_IF


// Position 2 Reached - Cylinder Timer OFF

IF NOT Solenoid2 THEN Timer2 :=0; END_IF


//Timer2 is for Monitoring Cylinder Work Position Time
WorkPositionErr_1SecPls(CLK := Pulse_1Sec);

IF Solenoid2 AND NOT Sensor2 AND WorkPositionErr_1SecPls.Q THEN 
	Timer2 := Timer2 + 1;
ELSE
	Timer2	:=0;
END_IF


//Generate Alarm for Work Position Sensor & Valve

IF Timer2 >= TimeOut2 AND NOT Sensor2 AND NOT Sensor1 THEN AlarmSensor2 :=1; END_IF
IF Timer2 >= TimeOut2 AND NOT Sensor2 AND Sensor1 THEN AlarmSolenoid2 :=1; END_IF


//Move "0" to Timer3 If anyone Sensor is not Sensing

IF NOT Sensor1 AND NOT Sensor2 THEN Timer3 :=0; END_IF


//Timer3 is for Monitoring Both Sensor ON Error
BothSensorErr_1SecPls (CLK := Pulse_1Sec);

 IF Sensor1 AND Sensor2 AND BothSensorErr_1SecPls.Q THEN
	 Timer3 := Timer3 + 1;
 ELSE
	 Timer3:=0;
 END_IF
 
 
 //Generate Alarm for Both Sensor ON Error
 
 IF Timer3 >= TimeOut3 THEN AllSignal :=1; END_IF
 
 
 //Reset the Valve when Operation Enable not Present
 
 IF NOT OperationEnable THEN
	 Solenoid1 :=0;
	 Solenoid2 :=0;
 END_IF

 
//Position 1 is Cylinder Home Position || Position 2 is Cylinder Work Position

Position1 := NOT AllSignal AND Sensor1 AND NOT Sensor2;
Position2 := NOT AllSignal AND Sensor2 AND NOT Sensor1; 

// ALARM RESET

IF ResetPB THEN
	
AlarmSensor1 								:= FALSE;
AlarmSensor2            					:= FALSE;
AlarmSolenoid1          					:= FALSE;
AlarmSolenoid2          					:= FALSE;
AllSignal               					:= FALSE;

END_IF


IF AlarmSensor1 OR AlarmSensor2 OR AlarmSolenoid1 OR AlarmSolenoid2 OR AllSignal THEN
		AlarmPresent						:= TRUE;
ELSE
		AlarmPresent						:= FALSE;
END_IF

END_FUNCTION_BLOCK

// ---- FB/Cylinder_Block_FOR_OP130.TcPOU
FUNCTION_BLOCK Cylinder_Block_FOR_OP130
VAR_INPUT
	Auto :BOOL;
	Manual :BOOL;
	ErrorActive :BOOL;
	ResetPB :BOOL;
	Sensor1 :BOOL;
	Sensor2 :BOOL;
	ManualPB1 :BOOL;
	ManualPB2 :BOOL;
	AutoCmd1 :BOOL;
	AutoCmd2 :BOOL;
	OperationEnable :BOOL;
	SafeHome :BOOL;
	SafeWork :BOOL;
	HomingCmd1 :BOOL;
	HomingCmd2 :BOOL;
	Pulse_1Sec :BOOL;
	BlinkingBit :BOOL;
	TimeOut1 :INT;
	TimeOut2 :INT;
	TimeOut3 :INT;
END_VAR
VAR_OUTPUT
	Solenoid1 :BOOL;
	Solenoid2 :BOOL;
	AlarmSensor1 :BOOL;
	AlarmSensor2 :BOOL;
	AlarmSolenoid1 :BOOL;
	AlarmSolenoid2 :BOOL;
	AllSignal :BOOL;
	AlarmPresent :BOOL;
	Position1 :BOOL;
	Position2 :BOOL;
	HomeSensorBlink :BOOL;
	WorkSensorBlink :BOOL;
END_VAR
VAR_IN_OUT
	Status :INT;
END_VAR
VAR
	Timer1 :INT;
	Timer2 :INT;
	Timer3 :INT;
	HomePositionErr_1SecPls :Tc2_Standard.R_TRIG;
	WorkPositionErr_1SecPls :Tc2_Standard.R_TRIG;
	BothSensorErr_1SecPls :Tc2_Standard.R_TRIG;
	Temp4 :BOOL;
END_VAR

Status:=0;

//Cylinder Moving to Home Position by Manual

IF ManualPB1 THEN
	IF NOT Manual THEN Status :=1; 
	ELSIF ManualPB2 THEN Status :=2; 
	ELSIF AllSignal THEN Status :=3;
	ELSIF NOT OperationEnable THEN Status :=9; 
	ELSIF Status =0 AND SafeHome THEN
		Solenoid1 :=1;
		Solenoid2 :=0;
	END_IF 
END_IF


//Cylinder Moving to Work Position by Manual

IF ManualPB2 THEN
	IF NOT Manual THEN Status :=1; 
	ELSIF ManualPB1 THEN Status :=2; 
	ELSIF AllSignal THEN Status :=3;
	ELSIF NOT OperationEnable THEN Status :=9; 
	ELSIF Status =0 AND SafeWork THEN
		Solenoid2 :=1;
		Solenoid1 :=0;
	END_IF 
END_IF


//Cylinder Moving to Home Position by Auto

IF AutoCmd1 THEN
	IF NOT Auto THEN Status :=5; 
	ELSIF AutoCmd2 THEN Status :=6;
	ELSIF ErrorActive THEN Status :=4; 
	ELSIF AllSignal THEN Status :=3;
	ELSIF NOT OperationEnable THEN Status :=9; 
	ELSIF Status =0 AND SafeHome THEN
		Solenoid1 :=1;
		Solenoid2 :=0;
	END_IF 
END_IF


//Cylinder Moving to Work Position by Auto

IF AutoCmd2 THEN
	IF NOT Auto THEN Status :=5; 
	ELSIF AutoCmd1 THEN Status :=6;
	ELSIF ErrorActive THEN Status :=4; 
	ELSIF AllSignal THEN Status :=3;
	ELSIF NOT OperationEnable THEN Status :=9; 
	ELSIF Status =0 AND SafeWork THEN
		Solenoid2 :=1;
		Solenoid1 :=0;
	END_IF 
END_IF


//Cylinder Moving to Home Position - Homing Cmd ON

IF HomingCmd1 THEN 
	IF AllSignal THEN Status :=3;
	ELSIF NOT OperationEnable THEN Status :=9; 
	ELSIF Status =0 AND SafeHome THEN
		Solenoid1 :=1;
		Solenoid2 :=0;
	END_IF 
END_IF
IF HomingCmd2 THEN 
	IF AllSignal THEN Status :=3;
	ELSIF NOT OperationEnable THEN Status :=9; 
	ELSIF Status =0 AND SafeHome THEN
		Solenoid2 :=1;
		Solenoid1 :=0;
	END_IF 
END_IF


// While Cylinder Moving Blinking IF Position Reached then Steady Indication

HomeSensorBlink := (Solenoid1 AND NOT Sensor1 AND BlinkingBit) OR Sensor1;
WorkSensorBlink := (Solenoid2 AND NOT Sensor2 AND BlinkingBit) OR Sensor2;


// Position 1 Reached - Cylinder Timer OFF

IF NOT Solenoid1 THEN Timer1 :=0; END_IF


//Timer1 is for Monitoring Cylinder Home Position Time
HomePositionErr_1SecPls(CLK := Pulse_1Sec);

IF Solenoid1 AND NOT Sensor1  AND HomePositionErr_1SecPls.Q THEN 
Timer1 := Timer1 + 1;
ELSE
Timer1:= 0;	
END_IF


//Generate Alarm for Home Position Sensor & Valve

IF Timer1 >= TimeOut1 AND NOT Sensor1 AND NOT Sensor2 THEN AlarmSensor1 :=1; END_IF
IF Timer1 >= TimeOut1 AND NOT Sensor1 AND Sensor2 THEN AlarmSolenoid1 :=1; END_IF


// Position 2 Reached - Cylinder Timer OFF

IF NOT Solenoid2 THEN Timer2 :=0; END_IF


//Timer2 is for Monitoring Cylinder Work Position Time
WorkPositionErr_1SecPls(CLK := Pulse_1Sec);

IF Solenoid2 AND NOT Sensor2 AND WorkPositionErr_1SecPls.Q THEN 
	Timer2 := Timer2 + 1;
ELSE
	Timer2:=0;
END_IF


//Generate Alarm for Work Position Sensor & Valve

IF Timer2 >= TimeOut2 AND NOT Sensor2 AND NOT Sensor1 THEN AlarmSensor2 :=1; END_IF
IF Timer2 >= TimeOut2 AND NOT Sensor2 AND Sensor1 THEN AlarmSolenoid2 :=1; END_IF


//Move "0" to Timer3 If anyone Sensor is not Sensing

IF NOT Sensor1 AND NOT Sensor2 THEN Timer3 :=0; END_IF


//Timer3 is for Monitoring Both Sensor ON Error
BothSensorErr_1SecPls (CLK := Pulse_1Sec);

 IF Sensor1 AND Sensor2 AND BothSensorErr_1SecPls.Q THEN
	 Timer3 := Timer3 + 1;
 END_IF
 
 
 //Generate Alarm for Both Sensor ON Error
 
 IF Timer3 >= TimeOut3 THEN AllSignal :=1; END_IF
 
 
 //Reset the Valve when Operation Enable not Present
 
 IF NOT OperationEnable THEN
	 Solenoid1 :=0;
	 Solenoid2 :=0;
 END_IF

 
//Position 1 is Cylinder Home Position || Position 2 is Cylinder Work Position

Position1 := NOT AllSignal AND Sensor1 AND NOT Sensor2;
Position2 := NOT AllSignal AND Sensor2 AND NOT Sensor1; 

// ALARM RESET

IF ResetPB THEN
	
AlarmSensor1 								:= FALSE;
AlarmSensor2            					:= FALSE;
AlarmSolenoid1          					:= FALSE;
AlarmSolenoid2          					:= FALSE;
AllSignal               					:= FALSE;

END_IF

END_FUNCTION_BLOCK

// ---- FB/Schunk/FB_Schunk.TcPOU
FUNCTION_BLOCK FB_Schunk
VAR_INPUT
iHW: 											ARRAY [0..8] OF WORD;
//i_b_moveToPosition:								BOOL;
i_b_moveRelativ:								BOOL;	
//i_b_reference:									BOOL;
i_b_ackError:									BOOL;
i_u_targetPos:									REAL;
i_u_targetVelocity:								REAL;
i_u_targetCurrent:								REAL;
i_u_targetAcceleration:							REAL;
i_u_targetJerk:									REAL;
i_b_ManualMode: 								BOOL;

END_VAR
VAR_IN_OUT
    stManualModeAxis  	: stManualModeAxis;
	i_b_reference:									BOOL;
	i_b_moveToPosition:								BOOL;
END_VAR
VAR_OUTPUT
Status: 										STRING;	
o_b_referenced:									BOOL;
o_b_reachedPos:									BOOL;	
o_u_actualPosition:								REAL;
o_b_error:										BOOL;
o_b_enable:										BOOL;
oHW:											ARRAY [0..11] OF WORD;

END_VAR
VAR
	
iProcessData:									UNION_iSchunkProcessData;
iStep:											ENUM_Schunk;
bError:											BOOL;

bHMFPErrorReset:								BOOL;
bHMFPManualErrorReset:							BOOL;
bHMFPHoming:									BOOL;
bHMFPMovePosition:								BOOL;
bHMFPMoveRelativ:								BOOL;
bHMFPAxisHomeDone:								BOOL;
bHMFPAxisPositionDone:							BOOL;
tonStateTimeOut: 								TON;


stat_commandReleaseA:							BOOL;
stat_commandReleaseB:							BOOL;
stat_oProcessData:								oSchunkProcessData;
stat_iProcessData:								iSchunkProcessData;

stat_targetVelocity:							REAL;
stat_targetPos:									REAL;

oProcessData:									UNION_oSchunkProcessData;
stat_newJob:									BOOL;
stat_HMnewJob:									BOOL;

END_VAR

VAR_TEMP
bFPnewJob:										BOOL;
bFPErrorReset: 									BOOL;
bFPManualErrorReset:							BOOL;
bFPHoming:										BOOL;
bFPMovePosition:								BOOL;
bFPMoveRelativ:									BOOL;
bTIN:											BOOL;
bFPAxisHomeDone:								BOOL;
bFPAxisPositionDone:							BOOL;
END_VAR


iProcessData.Schunk_in:= iHW;

stat_iProcessData.actualPos:= FC_Real_Convert(in:= iProcessData.iSchunk_ProcessData.actualPos);
stat_iProcessData.actualVelo:= FC_Real_Convert(in:= iProcessData.iSchunk_ProcessData.actualVelo);
stat_iProcessData.actualCurrent:= FC_Real_Convert(in:= iProcessData.iSchunk_ProcessData.actualCurrent);


// error bit
bError:= iProcessData.iSchunk_ProcessData.error;

// FP error reset
bFPErrorReset:= i_b_ackError AND NOT bHMFPErrorReset;
bHMFPErrorReset:= i_b_ackError;

bFPManualErrorReset:=stManualModeAxis.reset AND NOT bHMFPManualErrorReset;
bHMFPManualErrorReset:=stManualModeAxis.reset;

// FP homing
bFPHoming:= i_b_reference AND NOT bHMFPHoming;
bHMFPHoming:=i_b_reference;


// FP move position
bFPMovePosition:= i_b_moveToPosition AND NOT bHMFPMovePosition;
bHMFPMovePosition:= i_b_moveToPosition;

// FP move relativ
bFPMoveRelativ:= i_b_moveRelativ AND NOT bHMFPMoveRelativ;
bHMFPMoveRelativ:=i_b_moveRelativ;

// FP axis home done
bFPAxisHomeDone:=iProcessData.iSchunk_ProcessData.modulIsReferenced AND NOT bHMFPAxisHomeDone;
bHMFPAxisHomeDone:=iProcessData.iSchunk_ProcessData.modulIsReferenced;

// FP axis position done
bFPAxisPositionDone:=iProcessData.iSchunk_ProcessData.targetPosReached AND NOT bHMFPAxisPositionDone;
bHMFPAxisPositionDone:= iProcessData.iSchunk_ProcessData.targetPosReached;


// actual values 
o_u_actualPosition:= stat_iProcessData.actualPos;
stManualModeAxis.actualPosition := stat_iProcessData.actualPos;
stManualModeAxis.actualVelocity := stat_iProcessData.actualVelo;



// manual Mode
IF i_b_ManualMode THEN	
	stManualModeAxis.stationModeAutoManual:= FALSE;		
ELSE
	stManualModeAxis.jogPos := FALSE;
	stManualModeAxis.jogNeg := FALSE;
	stManualModeAxis.reset := FALSE;
	StManualModeAxis.openBrake:= FALSE;
	stManualModeAxis.homing:= FALSE;
	stManualModeAxis.moveAbsolute:= FALSE;
	stManualModeAxis.moveRelative:= FALSE;
	stManualModeAxis.moveVelocity:= FALSE;	
	stManualModeAxis.stationModeAutoManual:= TRUE;
END_IF


// velocity 
IF i_b_ManualMode THEN
	stat_targetVelocity:= stManualModeAxis.targetVelocity;
ELSE
	stat_targetVelocity:= i_u_targetVelocity;
END_IF

// Position
IF i_b_ManualMode THEN
	stat_targetPos:= stManualModeAxis.targetPositon;
ELSE
	stat_targetPos:= i_u_targetPos;
END_IF


stat_newJob:= FALSE;

stat_oProcessData.commandReleaseA:= FALSE;
stat_oProcessData.commandReleaseB:= FALSE;
stat_oProcessData.jerkActivate:= FALSE;
stat_oProcessData.currentActivate:= FALSE;
stat_oProcessData.accelerationActivate:=FALSE;
stat_oProcessData.velocityMove:= FALSE;
stat_oProcessData.moveToPosition:= FALSE;
stat_oProcessData.moveToRelativePosition:= FALSE;
stat_oProcessData.modulReference:= FALSE;
stat_oProcessData.restartModul:= FALSE;
stat_oProcessData.ackError:= FALSE;
stat_oProcessData.stop:= TRUE;
stat_oProcessData.fastStop:= TRUE;



CASE iStep OF
	

	ENUM_Schunk.Init:	//init all
	
						stat_newJob:= FALSE;

						stat_oProcessData.commandReleaseA:= FALSE;
						stat_oProcessData.commandReleaseB:= FALSE;
						stat_oProcessData.jerkActivate:= FALSE;
						stat_oProcessData.currentActivate:= FALSE;
						stat_oProcessData.accelerationActivate:=FALSE;
						stat_oProcessData.velocityMove:= FALSE;
						stat_oProcessData.moveToPosition:= FALSE;
						stat_oProcessData.moveToRelativePosition:= FALSE;
						stat_oProcessData.modulReference:= FALSE;
						stat_oProcessData.restartModul:= FALSE;
						stat_oProcessData.ackError:= FALSE;
						stat_oProcessData.stop:= TRUE;
						stat_oProcessData.fastStop:= TRUE;

						iStep:= ENUM_Schunk.Undefined;
		
	ENUM_Schunk.Undefined:
	
						IF bError THEN
							iStep:= ENUM_Schunk.Error;
						ELSE
							iStep:= ENUM_Schunk.Ready;
						END_IF
				
	ENUM_Schunk.Error:
	
						stat_newJob:= FALSE;
						stat_oProcessData.jerkActivate:= FALSE;
						stat_oProcessData.currentActivate:= FALSE;
						stat_oProcessData.accelerationActivate:=FALSE;
						stat_oProcessData.velocityMove:= FALSE;
						stat_oProcessData.moveToPosition:= FALSE;
						stat_oProcessData.moveToRelativePosition:= FALSE;
						o_b_referenced:= FALSE;
						o_b_reachedPos:= FALSE;
						o_b_error:= TRUE;
						
						IF bFPErrorReset OR  bFPManualErrorReset THEN
							iStep:= ENUM_Schunk.Reset;
						END_IF
						
	ENUM_Schunk.Reset:
	
						stat_oProcessData.ackError:= TRUE;
						stat_newJob:= TRUE;
						bTIN:=TRUE;
						o_b_error:= FALSE;
						
						IF NOT bError THEN
							bTIN:=FALSE;
							stat_oProcessData.ackError:= FALSE;
							stat_newJob:= FALSE;
							iStep:= ENUM_Schunk.Ready;
						ELSIF tonStateTimeOut.Q THEN
							bTIN:=FALSE;
							stat_oProcessData.ackError:= FALSE;
							stat_newJob:= FALSE;	
							iStep:= ENUM_Schunk.Error;
						END_IF
						tonStateTimeOut(IN:=bTIN,PT:=T#30S);
						
	ENUM_Schunk.Ready:
						//o_b_referenced:= FALSE;
						//o_b_reachedPos:= FALSE;
						
						IF bError THEN
							iStep:= ENUM_Schunk.Error;
						ELSIF bFPHoming OR stManualModeAxis.homing THEN
							iStep:= ENUM_Schunk.Homing;
						ELSIF bFPMovePosition OR stManualModeAxis.moveAbsolute THEN
							iStep:= ENUM_Schunk.MoveAbsolute;
						ELSIF bFPMoveRelativ OR stManualModeAxis.moveRelative THEN
							iStep:= ENUM_Schunk.MoveRelative;
						END_IF

	ENUM_Schunk.Homing:
	
					
						
						stat_oProcessData.modulReference:= TRUE;
						stat_newJob:= TRUE;
						bTIN:=TRUE;
						
						IF bError THEN
							stat_oProcessData.modulReference:= FALSE;
							bTIN:= FALSE;
							stat_newJob:= FALSE;
							iStep:= ENUM_Schunk.Error;
						ELSIF bFPAxisHomeDone THEN
							bTIN:= FALSE;
							stat_oProcessData.modulReference:= FALSE;
							stat_newJob:= FALSE;
							i_b_reference := FALSE;
							o_b_referenced:= TRUE;
							iStep:= ENUM_Schunk.Ready;
						ELSIF tonStateTimeOut.Q THEN
							bTIN:= FALSE;
							stat_oProcessData.modulReference:= FALSE;
							stat_newJob:= FALSE;
							iStep:= ENUM_Schunk.Error;
						END_IF
						tonStateTimeOut(IN:=bTIN,PT:=T#30S);
						
	ENUM_Schunk.MoveAbsolute:
	
					
	
						stat_oProcessData.currentActivate:= TRUE;
						stat_oProcessData.targetCurrent:= i_u_targetCurrent;
						stat_oProcessData.jerkActivate:= TRUE;
						stat_oProcessData.targetJerk:= i_u_targetJerk;
						stat_oProcessData.accelerationActivate:=TRUE;
						stat_oProcessData.targetAcc:= i_u_targetAcceleration;
						stat_oProcessData.velocityMove:= TRUE;
						stat_oProcessData.targetVelo:= stat_targetVelocity;
						stat_oProcessData.moveToPosition:= TRUE;
						stat_oProcessData.targetPos:= stat_targetPos;
						stat_newJob:= TRUE;					
						bTIN:=TRUE;
						IF bError THEN
							stat_oProcessData.currentActivate:=FALSE;
							stat_oProcessData.jerkActivate:=FALSE;
							stat_oProcessData.accelerationActivate:=FALSE;
							stat_oProcessData.velocityMove:=FALSE;
							stat_oProcessData.moveToPosition:=FALSE;
							bTIN:= FALSE;
							stat_newJob:= FALSE;
							iStep:= ENUM_Schunk.Error;
						ELSIF bFPAxisPositionDone THEN
							bTIN:= FALSE;
							stat_oProcessData.currentActivate:=FALSE;
							stat_oProcessData.jerkActivate:=FALSE;
							stat_oProcessData.accelerationActivate:=FALSE;
							stat_oProcessData.velocityMove:=FALSE;
							stat_oProcessData.moveToPosition:=FALSE;
							stat_newJob:= FALSE;
							i_b_moveToPosition:=FALSE;
							o_b_reachedPos:= TRUE;
							iStep:= ENUM_Schunk.Ready;
						ELSIF tonStateTimeOut.Q THEN
							bTIN:= FALSE;
							stat_oProcessData.currentActivate:=FALSE;
							stat_oProcessData.jerkActivate:=FALSE;
							stat_oProcessData.accelerationActivate:=FALSE;
							stat_oProcessData.velocityMove:=FALSE;
							stat_oProcessData.moveToPosition:=FALSE;
							stat_newJob:= FALSE;
							iStep:= ENUM_Schunk.Error;
						END_IF
						tonStateTimeOut(IN:=bTIN,PT:=T#30S);
						
	ENUM_Schunk.MoveRelative:
						
						
	
	
						stat_oProcessData.currentActivate:= TRUE;
						stat_oProcessData.targetCurrent:= i_u_targetCurrent;
						stat_oProcessData.jerkActivate:= TRUE;
						stat_oProcessData.targetJerk:= i_u_targetJerk;
						stat_oProcessData.accelerationActivate:=TRUE;
						stat_oProcessData.targetAcc:= i_u_targetAcceleration;
						stat_oProcessData.velocityMove:= TRUE;
						stat_oProcessData.targetVelo:= stat_targetVelocity;
						stat_oProcessData.moveToRelativePosition:= TRUE;
						stat_oProcessData.targetPos:= stat_targetPos;
						stat_newJob:= TRUE;	
						bTIN:=TRUE;
						
						IF bError THEN
							stat_oProcessData.currentActivate:=FALSE;
							stat_oProcessData.jerkActivate:=FALSE;
							stat_oProcessData.accelerationActivate:=FALSE;
							stat_oProcessData.velocityMove:=FALSE;
							stat_oProcessData.moveToPosition:=FALSE;
							bTIN:= FALSE;
							stat_newJob:= FALSE;
							iStep:= ENUM_Schunk.Error;
						ELSIF bFPAxisPositionDone THEN
							bTIN:= FALSE;
							stat_oProcessData.currentActivate:=FALSE;
							stat_oProcessData.jerkActivate:=FALSE;
							stat_oProcessData.accelerationActivate:=FALSE;
							stat_oProcessData.velocityMove:=FALSE;
							stat_oProcessData.moveToRelativePosition:=FALSE;
							stat_newJob:= FALSE;
							o_b_reachedPos:=TRUE;
							iStep:= ENUM_Schunk.Ready;
						ELSIF tonStateTimeOut.Q THEN
							bTIN:= FALSE;
							stat_oProcessData.currentActivate:=FALSE;
							stat_oProcessData.jerkActivate:=FALSE;
							stat_oProcessData.accelerationActivate:=FALSE;
							stat_oProcessData.velocityMove:=FALSE;
							stat_oProcessData.moveToPosition:=FALSE;
							stat_newJob:= FALSE;
							iStep:= ENUM_Schunk.Error;
						END_IF
						tonStateTimeOut(IN:=bTIN,PT:=T#30S);
END_CASE

// job

bFPnewJob:=stat_newJob AND NOT stat_HMnewJob;
stat_HMnewJob:=stat_newJob;

	IF bFPnewJob  THEN
		stat_commandReleaseA:= NOT stat_commandReleaseA;
		stat_oProcessData.commandReleaseA:= stat_commandReleaseA;
		stat_commandReleaseB:= NOT stat_commandReleaseA;
		stat_oProcessData.commandReleaseB:= stat_commandReleaseB;
		
		// Output
		oProcessData.oSchunk_ProcessData:= stat_oProcessData;
		oProcessData.oSchunk_ProcessData.targetPos:= FC_Real_Convert(in:= stat_oProcessData.targetPos );
		oProcessData.oSchunk_ProcessData.targetVelo:= FC_Real_Convert(in:=stat_oProcessData.targetVelo );
		oProcessData.oSchunk_ProcessData.targetCurrent:= FC_Real_Convert(in:=stat_oProcessData.targetCurrent );
		oProcessData.oSchunk_ProcessData.targetAcc:= FC_Real_Convert(in:=stat_oProcessData.targetAcc );
		oProcessData.oSchunk_ProcessData.targetJerk:= FC_Real_Convert(in:=stat_oProcessData.targetJerk );

	END_IF

	stManualModeAxis.axisState:= TO_STRING(iStep);
	//Status :=stManualModeAxis.axisState;
	oHW:=oProcessData.Schunk_out;
	
IF iHW[0].6 AND iHW[0].9 THEN
	o_b_reachedPos := TRUE ;
	Status :=stManualModeAxis.axisState;
ELSIF iHW[0].8 THEN
	Status:='Moving';
	o_b_reachedPos := FALSE;
END_IF

IF iHW[0].6 THEN
	o_b_enable := TRUE ;
ELSE
	o_b_enable := FALSE;
END_IF

END_FUNCTION_BLOCK

// ---- FB/Schunk/FC_Real_Convert.TcPOU
FUNCTION FC_Real_Convert : REAL
VAR_INPUT
	in	:REAL;
END_VAR
VAR
	uRealIn		:union_real;
	uRealOut	:union_real;
	
	
END_VAR

uRealIn.rREAL :=in;

uRealOut.aARRAY[0] := uRealIn.aARRAY[3];
uRealOut.aARRAY[1] := uRealIn.aARRAY[2];
uRealOut.aARRAY[2] := uRealIn.aARRAY[1];
uRealOut.aARRAY[3] := uRealIn.aARRAY[0];

FC_Real_Convert:=uRealOut.rREAL;

END_FUNCTION

// ---- POUs/Programs/OP10/OP10_AUTO.TcPOU
PROGRAM OP10_AUTO
VAR
	r1							: R_TRIG;	
	STEP_NO						: INT;
	STP_NO						: INT;
	AFT_GRP_HME					: TON;
	AFT_SRV_WRK					: TON;
	AFT_GRP_WRK					: TON;
	AFT_ROBO_CM_GRP_OPN			: TON;
	CMR_RSLT_DN					: TON;
	OP10_BODY_SING_HOME			: BOOL;
END_VAR

VAR PERSISTENT
	AFT_GRP_HME_TIME			: TIME;
	AFT_SRV_WRK_TIME			: TIME;
	AFT_GRP_WRK_TIME			: TIME;	
	AFT_ROBO_GRP_OPN			: TIME;
	OP10_COUNT					: DINT;
	OP10A_Auto_Status			: STRING;
	OP10B_Auto_Status			: STRING;
END_VAR



(*
IF  CHECK OR OP10A_AUTO_RUNNING OR OP10A_STEP_RUNNING OR OP10B_AUTO_RUNNING OR OP10B_STEP_RUNNING THEN

IF (OP10A_STRT_PB OR OP10B_STRT_PB OR CHECK)AND STEP_NO=0 THEN
	STEP_NO							:= 1;
	STP_NO							:= 1;
END_IF	


CASE STEP_NO OF
	
	1:	IF NOT END_OF_CYCLE THEN
		IF OP10_COMP_PICKED_1	THEN
		STEP_NO							:= 20;
		ELSE
		STEP_NO							:= 2;
		END_IF 
		ELSE
		STEP_NO							:= 0;		
		END_IF


	2:	IF I10_LH_LNR_TRK_BDY_PRSN_I1000_5 AND NOT (OP10A_ROBO_Gripper_Close AND OP10A_Rbt_In_Pick_Zone) 
			AND NOT (OP10B_ROBO_Gripper_Close AND OP10B_Rbt_In_Pick_Zone)THEN
		OP10_A_FRT_BDY_SING_HME			:= TRUE; 
		OP10_A_FRT_BDY_SING_WRK			:= FALSE;
		STEP_NO							:= 5;
		END_IF

	5: IF AFT_GRP_HME.Q THEN
		OP10_A_SRV_FST_BDYPCK_WRK		:= TRUE;
		STEP_NO							:= 10;	
		END_IF
	
	
	10: IF AFT_SRV_WRK.Q THEN
		OP10_A_FRT_BDY_SING_HME			:= FALSE; 
 	    OP10_A_FRT_BDY_SING_WRK			:= TRUE;
		OP10_COMP_PICKED_1				:= TRUE;
		STEP_NO							:= 15;
		END_IF
		
	15: IF AFT_GRP_WRK.Q THEN
		OP10_A_SRV_FST_BDYPCK_HME		:= TRUE;		
		STEP_NO							:= 20;
		END_IF	

	20:	IF OP10_SRV_FRST_PCKBDY_HME_FB THEN
													//		OP10_LH_CMP_RDY_PCK				:= TRUE;
		OP10A_SING_CMR_TRIG				:= TRUE;
		STEP_NO							:= 25;		
		END_IF
		
	25: CMR_RSLT_DN(IN:=(STEP_NO=25) AND NOT OP10A_SING_CAM_DN , PT:=T#1.5S , Q=> , ET=> );	
		IF CMR_RSLT_DN.Q THEN
		OP10A_SING_CMR_TRIG				:= FALSE;	
		STEP_NO							:= 20;	
		END_IF
		IF OP10A_SING_CAM_DN OR OP10A_SING_CAM_BYPASS THEN
		STEP_NO							:= 30;			
		END_IF
		
	30: IF OP10A_Body_OK OR OP10A_SING_CAM_BYPASS THEN
		STEP_NO							:= 35;
		END_IF
		IF OP10A_Body_NOK THEN
		OP10_COMP_PICKED_1				:= FALSE;
		STEP_NO							:= 1;
		END_IF
		
	(*35: 

	
		IF AFT_ROBO_CM_GRP_OPN.Q OR CHECK THEN

		END_IF*)
		

	500: OP10_COMP_PICKED_1				:= FALSE;
		OP10_A_FRT_BDY_SING_HME			:= TRUE; 
		OP10_A_SEC_BDY_SING_HME			:= TRUE; 
		OP10_A_FRT_BDY_SING_WRK			:= FALSE;
		OP10_A_SEC_BDY_SING_WRK			:= FALSE;
		OP10_LH_CMP_RDY_PCK				:= FALSE;
		OP10_RH_CMP_RDY_PCK				:= FALSE;		
		STEP_NO							:= 1;
	
END_CASE

		AFT_GRP_HME(IN:=(OP10_BDY_SING_FRT.Sensor1), PT:=AFT_GRP_HME_TIME, Q=> , ET=> );
		AFT_SRV_WRK(IN:=OP10_SRV_FRST_PCKBDY_WRK_FB, PT:=AFT_SRV_WRK_TIME , Q=> , ET=> );
		AFT_GRP_WRK(IN:= OP10_BDY_SING_FRT.Sensor2, PT:=AFT_GRP_WRK_TIME , Q=> , ET=> );
		AFT_ROBO_CM_GRP_OPN(IN:=(OP10A_ROBO_Gripper_Close AND OP10A_Rbt_In_Pick_Zone AND (OP10A_A_SRV_LH_GRPWRK_FB OR OP10A_BDY1_PCK_BYPAS) AND (OP10A_A_SRV_RH_GRPWRK_FB OR OP10A_BDY2_PCK_BYPAS))OR 
			(OP10B_ROBO_Gripper_Close AND OP10B_Rbt_In_Pick_Zone AND (OP10B_A_SRV_LH_GRPWRK_FB OR OP10B_BDY1_PCK_BYPAS)AND (OP10B_A_SRV_RH_GRPWRK_FB OR OP10B_BDY2_PCK_BYPAS)), PT:=AFT_ROBO_GRP_OPN, Q=> , ET=> );

CASE STP_NO OF

	1:	IF NOT END_OF_CYCLE THEN
		IF OP10_COMP_PICKED_2	THEN
		STEP_NO							:= 20;
		ELSE
		STEP_NO							:= 2;
		END_IF 
		ELSE
		STEP_NO							:= 0;		
		END_IF


	2:	IF I10_LH_LNR_TRK_BDY_PRSN_I1000_5 AND I10_RH_LNR_TRK_BDY_PRSN_I1000_6 AND NOT (OP10A_ROBO_Gripper_Close AND OP10A_Rbt_In_Pick_Zone) 
			AND NOT (OP10B_ROBO_Gripper_Close AND OP10B_Rbt_In_Pick_Zone)THEN
		OP10_A_FRT_BDY_SING_HME			:= TRUE; 
		OP10_A_SEC_BDY_SING_HME			:= TRUE; 
		OP10_A_FRT_BDY_SING_WRK			:= FALSE;
		OP10_A_SEC_BDY_SING_WRK			:= FALSE;
		STEP_NO							:= 5;
		END_IF

	5: IF AFT_GRP_HME.Q THEN
		OP10_A_SRV_FST_BDYPCK_WRK		:= TRUE;
		OP10_A_SRV_SCND_BDYPCK_WRK		:= TRUE;
		OP10_COMP_PICKED_2				:= TRUE;
		STEP_NO							:= 10;	
		END_IF
	
	
	10: IF AFT_SRV_WRK.Q THEN
		IF OP10_SRV_FRST_PCKBDY_WRK_FB THEN
		OP10_A_FRT_BDY_SING_HME			:= FALSE; 
 	    OP10_A_FRT_BDY_SING_WRK			:= TRUE;
		END_IF
		IF OP10_SRV_SCND_PCKBDY_WRK_FB THEN
		OP10_A_SEC_BDY_SING_HME			:= FALSE;
		OP10_A_SEC_BDY_SING_WRK			:= TRUE;
		END_IF	
		IF OP10_SRV_FRST_PCKBDY_WRK_FB AND OP10_SRV_SCND_PCKBDY_WRK_FB THEN
		STEP_NO							:= 15;	
		END_IF
		END_IF
		
	15: IF AFT_GRP_WRK.Q THEN
		OP10_A_SRV_SCND_BDYPCK_HME		:= TRUE;	
		OP10_A_SRV_FST_BDYPCK_HME		:= TRUE;	
		STEP_NO							:= 20;
		END_IF	

	20:	IF OP10_SRV_FRST_PCKBDY_HME_FB AND OP10_SRV_SCND_PCKBDY_HME_FB THEN
		OP10_LH_CMP_RDY_PCK				:= TRUE;
		OP10_RH_CMP_RDY_PCK				:= TRUE;
		IF AFT_ROBO_CM_GRP_OPN.Q OR CHECK THEN
		STEP_NO							:= 25;
		END_IF
		END_IF

	25: OP10_COMP_PICKED_2				:= FALSE;
		OP10_A_FRT_BDY_SING_HME			:= TRUE; 
		OP10_A_SEC_BDY_SING_HME			:= TRUE; 
		OP10_A_FRT_BDY_SING_WRK			:= FALSE;
		OP10_A_SEC_BDY_SING_WRK			:= FALSE;
		OP10_LH_CMP_RDY_PCK				:= FALSE;
		OP10_RH_CMP_RDY_PCK				:= FALSE;		
		STEP_NO							:= 1;



END_CASE

ELSE
		STEP_NO							:= 0;
		STP_NO							:= 0;
		OP10_A_SRV_FST_BDYPCK_WRK		:= FALSE;
		OP10_A_SRV_SCND_BDYPCK_WRK		:= FALSE;
		OP10_A_FRT_BDY_SING_HME			:= FALSE; 
		OP10_A_SEC_BDY_SING_HME			:= FALSE; 
		OP10_A_FRT_BDY_SING_WRK			:= FALSE;
		OP10_A_SEC_BDY_SING_WRK			:= FALSE;
		OP10_A_SRV_SCND_BDYPCK_HME		:= FALSE;	
		OP10_A_SRV_FST_BDYPCK_HME		:= FALSE;
END_IF


IF CHECK AND OP10_BODY_SING_HOME THEN
	OP10_A_SRV_SCND_BDYPCK_HME		:= (OP10_BDY_SING_FRT.Sensor1 AND OP10_BDY_SING_SEC.Sensor1) ;		
	OP10_A_SRV_FST_BDYPCK_HME	    := (OP10_BDY_SING_FRT.Sensor1 AND OP10_BDY_SING_SEC.Sensor1) ;
	OP10_A_SRV_FST_BDYPCK_WRK		:= FALSE;
	OP10_A_SRV_SCND_BDYPCK_WRK		:= FALSE;
	OP10_A_FRT_BDY_SING_HME			:= TRUE; 
 	OP10_A_FRT_BDY_SING_WRK			:= FALSE;
	OP10_A_SEC_BDY_SING_HME			:= TRUE;
	OP10_A_SEC_BDY_SING_WRK			:= FALSE;	
	STEP_NO							:= 1;
END_IF








r1(CLK:=OP10_SRV_FRST_PCKBDY_HME_FB AND OP10_SRV_SCND_PCKBDY_HME_FB , Q=> );
IF r1.Q THEN
	OP10_COUNT:=OP10_COUNT+1;
END_IF

*)

END_PROGRAM

// ---- POUs/Programs/OP10/OP10_Body_Camera_Seq.TcPOU
PROGRAM OP10_Body_Camera_Seq
VAR
	Toggle_Pos_LH_Empty : R_TRIG;
	Toggle_Neg_LH_Empty : F_TRIG;
	Toggle_Pos_RH_Empty : R_TRIG;
	Toggle_Neg_RH_Empty : F_TRIG;
	LH_Empty_Cam_Completed : BOOL;
	RH_Empty_Cam_Completed : BOOL;
	Body_Singulation_Cam_Seq: INT;
END_VAR

Toggle_Pos_LH_Empty(CLK:=OP10A_Camera_FB.OP10A_Empty_Cam_1_Inspection_Status.Inspection_Completed);
Toggle_Neg_LH_Empty(CLK:=OP10A_Camera_FB.OP10A_Empty_Cam_1_Inspection_Status.Inspection_Completed);
Toggle_Pos_RH_Empty(CLK:=OP10B_Camera_FB.OP10B_Empty_Cam_2_Inspection_Status.Inspection_Completed);
Toggle_Neg_RH_Empty(CLK:=OP10B_Camera_FB.OP10B_Empty_Cam_2_Inspection_Status.Inspection_Completed);

IF Toggle_Pos_LH_Empty.Q OR Toggle_Pos_LH_Empty.Q THEN
	LH_Empty_Cam_Completed:=1;	
END_IF
IF Toggle_Pos_RH_Empty.Q OR Toggle_Pos_RH_Empty.Q THEN
	RH_Empty_Cam_Completed:=1;	
END_IF

IF OP10A_AUTO_RUNNING AND Body_Singulation_Cam_Seq=0 OR (NOT OP10A_Empty_Cam_1_Camera_Online OR NOT OP10B_Empty_Cam_2_Camera_Online) THEN
	Body_Singulation_Cam_Seq:=10;
END_IF  

CASE Body_Singulation_Cam_Seq OF
	10: 	OP10A_Body_OK			  := 0;
            OP10A_Body_NOK			  := 0;
            OP10B_Body_OK			  := 0;
            OP10B_Body_NOK			  := 0;
            OP10A_Body_Window_OK	  := 0;
            OP10A_Body_Window_NOK	  := 0;
            OP10B_Body_Window_OK	  := 0;
            OP10B_Body_Window_NOK	  := 0;	
			LH_Empty_Cam_Completed    :=0;
			RH_Empty_Cam_Completed    :=0;		
			OP10_Body_Empty_Cam_Done  :=0;
			OP10_Body_Gripping_Done   :=0;
			Body_Singulation_Cam_Seq	  :=11;	
	
	11: IF (OP10_Empty_Camera_Trigger AND (NOT OP10_Body_Empty_Cam_Done)) THEN
			OP10A_Empty_Cam_1_Camera_Trigger:=1;
			OP10B_Empty_Cam_2_Camera_Trigger:=1;
			Body_Singulation_Cam_Seq	:=15;	
		END_IF

	15:	IF LH_Empty_Cam_Completed AND RH_Empty_Cam_Completed THEN
			OP10A_Empty_Cam_1_Camera_Trigger :=0;
			OP10B_Empty_Cam_2_Camera_Trigger :=0;
			OP10_Empty_Camera_Trigger :=0;
			Body_Singulation_Cam_Seq  :=25;
		END_IF  
	   
	25: IF OP10A_Camera_FB.OP10A_Empty_Cam_1_Result[0]=1 AND OP10B_Camera_FB.OP10B_Empty_Cam_2_Result[0]=1 THEN
			OP10A_Body_Window_OK 		:=1;
			OP10B_Body_Window_OK		:=1;
			OP10_Body_Empty_Cam_Done    :=1;
			Body_Singulation_Cam_Seq 	:=30;
		ELSIF OP10A_Camera_FB.OP10A_Empty_Cam_1_Result[0]<>1 AND OP10B_Camera_FB.OP10B_Empty_Cam_2_Result[0]=1 THEN	
			OP10A_Body_Window_NOK 		:=1;
			OP10B_Body_Window_OK		:=1;
			OP10_Body_Empty_Cam_Done    :=1;
			Body_Singulation_Cam_Seq    :=30;
		ELSIF OP10A_Camera_FB.OP10A_Empty_Cam_1_Result[0]=1 AND OP10B_Camera_FB.OP10B_Empty_Cam_2_Result[0]<>1 THEN			
			OP10A_Body_Window_OK 		:=1;
			OP10B_Body_Window_NOK		:=1;
			OP10_Body_Empty_Cam_Done    :=1;
			Body_Singulation_Cam_Seq    :=30;			
		ELSIF  OP10A_Camera_FB.OP10A_Empty_Cam_1_Result[0]<>1 AND OP10B_Camera_FB.OP10B_Empty_Cam_2_Result[0]<>1 THEN
			OP10A_Body_Window_NOK 		:=1;
			OP10B_Body_Window_NOK		:=1;
			OP10_Body_Empty_Cam_Done    :=1;
			Body_Singulation_Cam_Seq    :=30;	
		END_IF	
			
   30:  IF OP10_Body_Gripping_Done THEN
			Body_Singulation_Cam_Seq   :=10;
		END_IF	
   	    
END_CASE

END_PROGRAM

// ---- FB/Scanner/Scanner.TcPOU
FUNCTION_BLOCK Scanner
VAR_INPUT
	Acquisition_Status	: Acquisition_Status_Scanner;
	Result_Status		: Result_Status;
	Result_Data_Register: Result_Data_Register;
	Res_Data			: ARRAY[0..MAX_STRING_LENGTH] OF BYTE;
	reset				: BOOL;
END_VAR

VAR_OUTPUT
	Acquisition_Control	: Acquisition_Control_Scanner;
	Result_Control		: Result_Control_Scanner;
	Result_ID           : UINT;
	Read_Done			: BOOL;
	Busy				: BOOL;
	Result				: T_MaxString;
	No_Read				: BOOL;
	Error				: BOOL;
END_VAR

VAR_IN_OUT
	Scan_Start			: BOOL;
END_VAR

VAR
	trigger      : R_TRIG;
	rst		     : R_TRIG;
	okay	     : R_TRIG;
	ack			 : R_TRIG;
	i		     : INT ;
	in		     : ARRAY[0..MAX_STRING_LENGTH] OF BYTE;
	ok		     : BOOL;
	nok		     : BOOL;
	temp	     : UINT;	
	Scanner_Read : INT;
END_VAR


trigger(CLK:=Scan_Start);
rst(CLK:=reset);
okay(CLK:=Result_Status.Result_Available);
ack(CLK:=Result_Control.Result_acknowledge);
Busy:=Acquisition_Status.Acquiring;
Error:=Result_Status.Set_When_fault_Occur;

IF NOT Result_Status.Set_When_fault_Occur THEN
	IF NOT Acquisition_Control.Trigger_Enable THEN
		Acquisition_Control.Trigger_Enable:=1;
	END_IF
	IF trigger.Q=TRUE AND Acquisition_Control.Trigger_Enable THEN
		Acquisition_Control.Trigger:=1;
	END_IF
	IF okay.Q THEN
		Acquisition_Control.Trigger:=0;
	END_IF
	Result_ID:=Result_Data_Register.Result_ID;
END_IF

IF Result_Data_Register.Result_code=0 AND Scan_Start THEN
	Result:='';
	No_Read:=TRUE;
	Scan_Start:=0;
	nok:=1;ok:=0;
	Result_Control.Result_Acknowledge:=TRUE;
ELSIF Result_Data_Register.Result_Code=1 AND Scan_Start THEN
	ok:=1;nok:=0;
	Scan_Start:=0;
	temp:=Result_Data_Register.Result_ID;
END_IF

IF Result_Status.Result_available AND ok AND NOT Result_Status.Set_When_fault_Occur  AND NOT Busy AND (temp<>Result_Data_Register.Result_ID) THEN
	FOR i:=0 TO 245 DO
		in[i]:=Res_Data[i];
    END_FOR
	Result:=BYTEARR_TO_MAXSTRING(in:=in);
	No_Read:=FALSE;
	Read_Done:=TRUE;
	temp:=Result_Data_Register.Result_ID;
	Result_Control.Result_acknowledge:=TRUE;
END_IF

IF rst.Q=TRUE OR BUSY THEN
	No_Read:=FALSE;
    Read_Done:=FALSE;
END_IF

IF ack.Q THEN
   Result_Control.Result_acknowledge:=FALSE;
END_IF

END_FUNCTION_BLOCK

// ---- POU1/Axis_Position_Bias.TcPOU
PROGRAM Axis_Position_Bias
VAR
	bSet_Encoder_Zero: BOOL;
	bSet_Encoder_Zero_Rtrig: R_trig;
	Step: INT;
	ADSREAD_set_val: ADSREAD;
	FB_GetLocalAmsNetId_system: FB_GetLocalAmsNetId;
	lrRead_set_Value: LREAL;
	stAxis:AXIS_REF;
	
	ADSWRITE_Set_Val: ADSWRITE;
	
	tDummy: Ton;
	bRead_set_Value: BOOL;
	bWrite_set_Value: BOOL;
	bHome_ref_done: BOOL;
	MC_Power1: MC_Power;
	bEnable: BOOL;
	TRIAL: BOOL;
	F_TRIG1: F_TRIG;
	home_pressed: BOOL;
	
END_VAR

VAR PERSISTENT
	aa: DINT;
lrWrite_set_Value: LREAL;
HOMING_VALUE: LREAL;
END_VAR

bSet_Encoder_Zero:=NOT TRIAL OR home_pressed;

bSet_Encoder_Zero_Rtrig.CLK:=bSet_Encoder_Zero;
bSet_Encoder_Zero_Rtrig();

IF bSet_Encoder_Zero_Rtrig.Q THEN Step :=10; END_IF

CASE Step OF 
10:
	lrRead_set_Value:=0; lrWrite_set_Value:=0; bRead_set_Value:=FALSE; bWrite_set_Value :=FALSE; 
	Step:=Step+10;
20:
	lrWrite_set_Value:=0; bWrite_set_Value :=TRUE; 
	tDummy.IN:=TRUE;
	IF tDummy.Q THEN tDummy.IN:=FALSE ; bWrite_set_Value := FALSE;Step:= step+10; END_IF
30:	IF home_pressed THEN
	lrWrite_set_Value:= stAxis.NcToPlc.ActPos * -1;
	ELSE
	 lrWrite_set_Value:=HOMING_VALUE;
	END_IF;
	Step:= step+10;
40:
	bWrite_set_Value := TRUE; tDummy.IN:=TRUE;
	IF tDummy.Q THEN tDummy.IN:=FALSE ;Step:= step+10; bWrite_set_Value := FALSE; END_IF
	IF ADSWRITE_Set_Val.ERR  THEN bWrite_set_Value := FALSE;tDummy.IN:=FALSE; Step:=10; END_IF
50:
	IF (LREAL_TO_INT(stAxis.NcToPlc.ActPos*10)=0 OR (lrWrite_set_Value=HOMING_VALUE)) AND ( home_pressed OR NOT TRIAL) THEN
		bHome_ref_done:=TRUE;	step:=99; bSet_Encoder_Zero:=FALSE;
	ELSE
 		step:=10;
END_IF 
	
END_CASE

FB_GetLocalAmsNetId_system.bExecute:=TRUE;
FB_GetLocalAmsNetId_system();

ADSWRITE_Set_Val(
	NETID:=FB_GetLocalAmsNetId_system.AddrString , 
	PORT:=501 , 	
	IDXGRP:=16#5006, 	
	IDXOFFS:=16#07,  
	LEN:= SIZEOF(lrWrite_set_Value), 
	SRCADDR:= ADR(lrWrite_set_Value) , 
	WRITE:=bWrite_set_Value ,   	    
	TMOUT:=T#500MS , 
	BUSY=> ,  
	ERR=> , 	
	ERRID=> );	

tDummy.PT:=T#20MS;
tDummy();	
	
(*MC_Power1(
	Axis:=stAxis, 
	Enable:=bEnable AND NOT home_pressed, 
	Enable_Positive:= 1, 
	Enable_Negative:= 1, 
	Override:=100 , 
	BufferMode:= , 
	Options:= , 
	Status=> , 
	Busy=> , 
	Active=> , 
	Error=> , 
	ErrorID=> );*)

TRIAL := (step=99);

IF (lrWrite_set_Value<>HOMING_VALUE)AND(step=99)THEN
	HOMING_VALUE:=lrWrite_set_Value;
END_IF

END_PROGRAM

// ---- POUs/GENERAL/MODE_SELECTION.TcPOU
PROGRAM MODE_SELECTION
VAR
		
END_VAR

// MODE FUNTIONAL BLOCK

FB_MODE_BLOCK(
	ModeWord:= MODE_WORD, 
	HomeConditionOK:= ALL_STN_IN_HOME, 
	OperationEnable:= SAFE_TO_WORK, 
	StartPB:= START_PB , 
	SafetyAndNOError:= , 
	ModeAck:=MODE_CHANGE_ACK, 
	HomingINProgress:= , 
	TempHomeOK:= , 
	ResetPB:= RESET_PB, 
	AutoSelected=> AUTO_SELECTED, 
	ManualSelected=> MANUAL_SELECTED, 
	StepSelected=> STEP_SELECTED, 
	ModeSelAck_Indication=> , 
	StatusDisplay=> , 
	AutoRunning:= AUTO_RUNNING, 
	StepRunning:= STEP_RUNNING, 
	StartEnable:= START_ENABLE, 
	MachineStop:= MACHINE_STOP);

END_PROGRAM

// ---- POUs/Programs/offline testing/cylinder_3_pos.TcPOU
FUNCTION_BLOCK cylinder_3_pos
VAR_INPUT
	en_in: BOOL;
	error_bit: BOOL;
	cylinder_work_coil:BOOL;
	cylinder_home_coil:BOOL;
	cylinder_mid_coil :BOOL;
	delay_1: LTIME;
	delay_2: LTIME;
	delay_3: LTIME;
	
END_VAR
VAR_OUTPUT
	en_out: BOOL;
	cylinder_work_fb:BOOL;
	cylinder_home_fb:BOOL;
	cylinder_mid_fb:BOOL;
	delay_display_1: LTIME;
	delay_display_2: LTIME;
	delay_display_3: LTIME;
END_VAR
VAR
	sensor_delay_1: LTON;
	sensor_delay_2: LTON;
	sensor_delay_3: LTON;
	

	
END_VAR
VAR_IN_OUT
	
END_VAR
VAR // added by the converter: edge detectors and wires of the graphical bodies
    _w1, _w2, _w3 : BOOL;
END_VAR

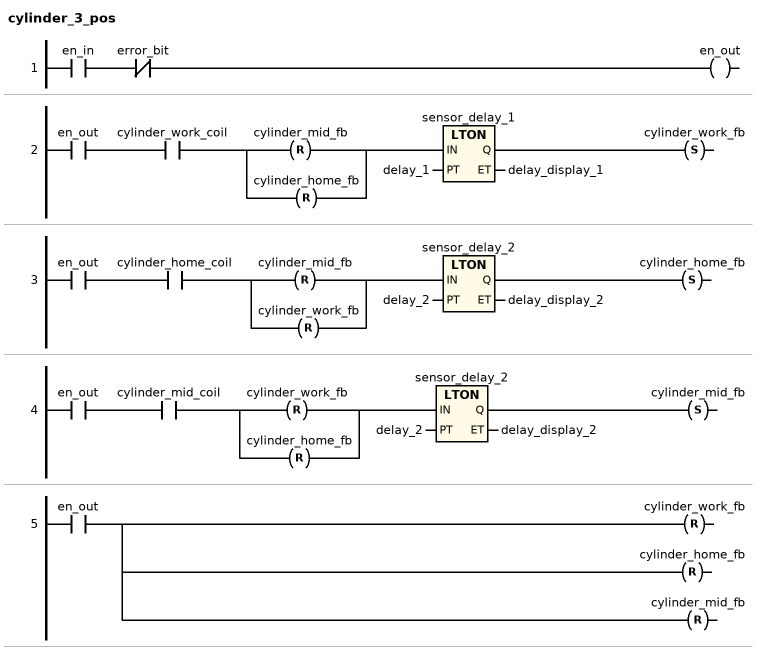
// NETWORK 1
en_out := en_in AND NOT error_bit;

// NETWORK 2
_w1 := en_out AND cylinder_work_coil;
cylinder_mid_fb R= _w1;
cylinder_home_fb R= _w1;
sensor_delay_1(IN := _w1, PT := delay_1, ET => delay_display_1); // LTON
cylinder_work_fb S= sensor_delay_1.Q;

// NETWORK 3
_w2 := en_out AND cylinder_home_coil;
cylinder_mid_fb R= _w2;
cylinder_work_fb R= _w2;
sensor_delay_2(IN := _w2, PT := delay_2, ET => delay_display_2); // LTON
cylinder_home_fb S= sensor_delay_2.Q;

// NETWORK 4
_w3 := en_out AND cylinder_mid_coil;
cylinder_work_fb R= _w3;
cylinder_home_fb R= _w3;
sensor_delay_2(IN := _w3, PT := delay_2, ET => delay_display_2); // LTON
cylinder_mid_fb S= sensor_delay_2.Q;

// NETWORK 5
cylinder_work_fb R= en_out;
cylinder_home_fb R= en_out;
cylinder_mid_fb R= en_out;

END_FUNCTION_BLOCK

// ---- POUs/Programs/offline testing/Cylinder_Block_v1.TcPOU
FUNCTION_BLOCK Cylinder_Block_v1
VAR_INPUT
	Auto :BOOL;
	Manual :BOOL;
	ErrorActive :BOOL;
	ResetPB :BOOL;
	Sensor1 :BOOL;
	Sensor2 :BOOL;
	ManualPB1 :BOOL;
	ManualPB2 :BOOL;
	AutoCmd1 :BOOL;
	AutoCmd2 :BOOL;
	OperationEnable :BOOL;
	SafeHome :BOOL;
	SafeWork :BOOL;
	HomingCmd1 :BOOL;
	Pulse_1Sec :BOOL;
	BlinkingBit :BOOL;
	TimeOut1 :INT;
	TimeOut2 :INT;
	TimeOut3 :INT;
END_VAR
VAR_OUTPUT
	Solenoid1 :BOOL;
	Solenoid2 :BOOL;
	AlarmSensor1 :BOOL;
	AlarmSensor2 :BOOL;
	AlarmSolenoid1 :BOOL;
	AlarmSolenoid2 :BOOL;
	AllSignal :BOOL;
	AlarmPresent :BOOL;
	Position1 :BOOL;
	Position2 :BOOL;
	HomeSensorBlink :BOOL;
	WorkSensorBlink :BOOL;
END_VAR
VAR_IN_OUT
	Status :INT;
END_VAR
VAR
	Timer1 :INT;
	Timer2 :INT;
	Timer3 :INT;
	HomePositionErr_1SecPls :Tc2_Standard.R_TRIG;
	WorkPositionErr_1SecPls :Tc2_Standard.R_TRIG;
	BothSensorErr_1SecPls :Tc2_Standard.R_TRIG;
	Temp4 :BOOL;
END_VAR
VAR_INPUT
	offline_bit: BOOL;
	error_bit: BOOL;
	cylinder_mid_coil :BOOL;
	delay_1: TIME;
	delay_2: TIME;
	delay_3: TIME;
	
END_VAR
VAR_OUTPUT

END_VAR
VAR
	en_out: BOOL;
	cylinder_mid_fb :BOOL;
	sensor_delay_1: TON;
	sensor_delay_2: TON;
	sensor_delay_3: TON;

END_VAR
VAR_IN_OUT
	
END_VAR



//Cylinder Moving to Home Position by Manual

IF ManualPB1 THEN
	IF NOT Manual THEN Status :=1; 
	ELSIF ManualPB2 THEN Status :=2; 
	ELSIF AllSignal THEN Status :=3;
	ELSIF NOT OperationEnable THEN Status :=9; 
	ELSIF Status =0 AND SafeHome THEN
		Solenoid1 :=1;
		Solenoid2 :=0;
	END_IF 
END_IF


//Cylinder Moving to Work Position by Manual

IF ManualPB2 THEN
	IF NOT Manual THEN Status :=1; 
	ELSIF ManualPB1 THEN Status :=2; 
	ELSIF AllSignal THEN Status :=3;
	ELSIF NOT OperationEnable THEN Status :=9; 
	ELSIF Status =0 AND SafeWork THEN
		Solenoid2 :=1;
		Solenoid1 :=0;
	END_IF 
END_IF


//Cylinder Moving to Home Position by Auto

IF AutoCmd1 THEN
	IF NOT Auto THEN Status :=5; 
	ELSIF AutoCmd2 THEN Status :=6;
	ELSIF ErrorActive THEN Status :=4; 
	ELSIF AllSignal THEN Status :=3;
	ELSIF NOT OperationEnable THEN Status :=9; 
	ELSIF Status =0 AND SafeHome THEN
		Solenoid1 :=1;
		Solenoid2 :=0;
	END_IF 
END_IF


//Cylinder Moving to Work Position by Auto

IF AutoCmd2 THEN
	IF NOT Auto THEN Status :=5; 
	ELSIF AutoCmd1 THEN Status :=6;
	ELSIF ErrorActive THEN Status :=4; 
	ELSIF AllSignal THEN Status :=3;
	ELSIF NOT OperationEnable THEN Status :=9; 
	ELSIF Status =0 AND SafeWork THEN
		Solenoid2 :=1;
		Solenoid1 :=0;
	END_IF 
END_IF


//Cylinder Moving to Home Position - Homing Cmd ON

IF HomingCmd1 THEN 
	IF AllSignal THEN Status :=3;
	ELSIF NOT OperationEnable THEN Status :=9; 
	ELSIF Status =0 AND SafeHome THEN
		Solenoid1 :=1;
		Solenoid2 :=0;
	END_IF 
END_IF


// While Cylinder Moving Blinking IF Position Reached then Steady Indication

HomeSensorBlink := (Solenoid1 AND NOT Sensor1 AND BlinkingBit) OR Sensor1;
WorkSensorBlink := (Solenoid2 AND NOT Sensor2 AND BlinkingBit) OR Sensor2;


// Position 1 Reached - Cylinder Timer OFF

IF NOT Solenoid1 THEN Timer1 :=0; END_IF


//Timer1 is for Monitoring Cylinder Home Position Time
HomePositionErr_1SecPls(CLK := Pulse_1Sec);

IF Solenoid1 AND HomePositionErr_1SecPls.Q THEN 
Timer1 := Timer1 + 1;
END_IF


//Generate Alarm for Home Position Sensor & Valve

IF Timer1 >= TimeOut1 AND NOT Sensor1 AND NOT Sensor2 THEN AlarmSensor1 :=1; END_IF
IF Timer1 >= TimeOut1 AND NOT Sensor1 AND Sensor2 THEN AlarmSolenoid1 :=1; END_IF


// Position 2 Reached - Cylinder Timer OFF

IF NOT Solenoid2 THEN Timer2 :=0; END_IF


//Timer2 is for Monitoring Cylinder Work Position Time
WorkPositionErr_1SecPls(CLK := Pulse_1Sec);

IF Solenoid2 AND WorkPositionErr_1SecPls.Q THEN 
	Timer2 := Timer2 + 1;
END_IF


//Generate Alarm for Work Position Sensor & Valve

IF Timer2 >= TimeOut2 AND NOT Sensor2 AND NOT Sensor1 THEN AlarmSensor2 :=1; END_IF
IF Timer2 >= TimeOut2 AND NOT Sensor2 AND Sensor1 THEN AlarmSolenoid2 :=1; END_IF


//Move "0" to Timer3 If anyone Sensor is not Sensing

IF NOT Sensor1 AND NOT Sensor2 THEN Timer3 :=0; END_IF


//Timer3 is for Monitoring Both Sensor ON Error
BothSensorErr_1SecPls (CLK := Pulse_1Sec);

 IF Sensor1 AND Sensor2 AND BothSensorErr_1SecPls.Q THEN
	 Timer3 := Timer3 + 1;
 END_IF
 
 
 //Generate Alarm for Both Sensor ON Error
 
 IF Timer3 >= TimeOut3 THEN AllSignal :=1; END_IF
 
 
 //Reset the Valve when Operation Enable not Present
 
 IF NOT OperationEnable THEN
	 Solenoid1 :=0;
	 Solenoid2 :=0;
 END_IF

 
//Position 1 is Cylinder Home Position || Position 2 is Cylinder Work Position
 
 

IF NOT  en_out THEN
	Position1 := NOT AllSignal AND Sensor1 AND NOT Sensor2;
    Position2 := NOT AllSignal AND Sensor2 AND NOT Sensor1;
	
END_IF

// validation offline

// timer inputs
sensor_delay_1.PT :=delay_1;
sensor_delay_2.PT :=delay_2;
sensor_delay_3.PT :=delay_3;

// offline test bit and error bit check
IF offline_bit AND NOT error_bit THEN
	en_out:=TRUE;
END_IF

// work feedback logic
IF  en_out AND ManualPB2 OR AutoCmd2  THEN
	sensor_delay_1.IN:=TRUE;
	Position1        :=FALSE;
	cylinder_mid_fb  :=FALSE;
	IF sensor_delay_1.Q THEN
		Position2:=TRUE;
	END_IF
END_IF

IF NOT ManualPB2 OR NOT AutoCmd2 THEN
	sensor_delay_1.IN:=FALSE;
END_IF

// home feedback logic
IF  en_out AND AutoCmd1 OR ManualPB1 OR HomingCmd1 THEN
	sensor_delay_2.IN:=TRUE;
	Position2        :=FALSE;
	cylinder_mid_fb  :=FALSE;
	IF sensor_delay_1.Q THEN
		Position1    :=TRUE;
	END_IF
END_IF

IF NOT AutoCmd1 OR NOT ManualPB1 OR NOT HomingCmd1 THEN
	sensor_delay_2.IN:=FALSE;
END_IF

// mid feedback logic
IF  en_out AND cylinder_mid_coil THEN
	sensor_delay_3.IN:=TRUE;
	Position1 :=FALSE;
	Position2  :=FALSE;
	IF sensor_delay_3.Q THEN
		cylinder_mid_fb:=TRUE;
	END_IF
END_IF

IF NOT cylinder_mid_coil THEN
	sensor_delay_3.IN:=FALSE;
END_IF

END_FUNCTION_BLOCK

// ---- POUs/Programs/offline testing/cylinder_validation_st.TcPOU
FUNCTION_BLOCK cylinder_validation_st
VAR_INPUT
	en_in: BOOL;
	error_bit: BOOL;
	cylinder_work_coil:BOOL;
	cylinder_home_coil:BOOL;
	cylinder_mid_coil :BOOL;
	delay_1: TIME;
	delay_2: TIME;
	delay_3: TIME;
	
END_VAR
VAR_OUTPUT
	en_out: BOOL;
	cylinder_work_fb:BOOL;
	cylinder_home_fb:BOOL;
	cylinder_mid_fb :BOOL;
	delay_display_1 : TIME;
	delay_display_2 : TIME;
	delay_display_3 : TIME;
END_VAR
VAR
	sensor_delay_1: TON;
	sensor_delay_2: TON;
	sensor_delay_3: TON;
	tim1 : ton;

	
END_VAR
VAR_IN_OUT
	
END_VAR

// cylinder validation block
// timer inputs
sensor_delay_1.PT :=delay_1;
sensor_delay_2.PT :=delay_2;
sensor_delay_3.PT :=delay_3;

// offline test bit and error bit check
IF en_in AND NOT error_bit THEN
	en_out:=TRUE;
END_IF

// work feedback logic
IF  en_out AND cylinder_work_coil THEN
	sensor_delay_1.IN:=TRUE;
	cylinder_home_fb :=FALSE;
	cylinder_mid_fb  :=FALSE;
	IF sensor_delay_1.Q THEN
		cylinder_work_fb:=TRUE;
	END_IF
END_IF

IF NOT cylinder_work_coil THEN
	sensor_delay_1.IN:=FALSE;
END_IF

// home feedback logic
IF  en_out AND cylinder_home_coil THEN
	sensor_delay_2.IN:=TRUE;
	cylinder_work_fb :=FALSE;
	cylinder_mid_fb  :=FALSE;
	IF sensor_delay_1.Q THEN
		cylinder_home_fb:=TRUE;
	END_IF
END_IF

IF NOT cylinder_home_coil THEN
	sensor_delay_2.IN:=FALSE;
END_IF

// mid feedback logic
IF  en_out AND cylinder_mid_coil THEN
	sensor_delay_3.IN:=TRUE;
	cylinder_work_fb :=FALSE;
	cylinder_home_fb  :=FALSE;
	IF sensor_delay_3.Q THEN
		cylinder_mid_fb:=TRUE;
	END_IF
END_IF

IF NOT cylinder_mid_coil THEN
	sensor_delay_3.IN:=FALSE;
END_IF

END_FUNCTION_BLOCK

// ---- POUs/Programs/offline testing/offline_fb.TcPOU
FUNCTION_BLOCK offline_fb
VAR
	cylinder_1: cylinder_2_pos;
	cylinder_2: cylinder_2_pos;
	cylinder_3: cylinder_2_pos;
	cylinder_4: cylinder_2_pos;
	cylinder_5: cylinder_2_pos;
	cylinder_6: cylinder_2_pos;
	cylinder_7: cylinder_2_pos;
	cylinder_8: cylinder_2_pos;
	cylinder_9: cylinder_2_pos;
	cylinder_10: cylinder_2_pos;
	servo_1: servo;
	servo_2: servo;
	servo_3: servo;
	servo_4: servo;
	servo_5: servo;
	servo_6: servo;
	servo_7: servo;
	servo_8: servo;
	servo_9: servo;
	servo_10: servo;
END_VAR

VAR_OUTPUT
	
	// cylinder out
	
cyl_work_fb_1   :BOOL;
cyl_home_fb_1   :BOOL;
cyl_work_fb_2   :BOOL;
cyl_home_fb_2   :BOOL;
cyl_work_fb_3   :BOOL;
cyl_home_fb_3   :BOOL;
cyl_work_fb_4   :BOOL;
cyl_home_fb_4   :BOOL;
cyl_work_fb_5   :BOOL;
cyl_home_fb_5   :BOOL;
cyl_work_fb_6   :BOOL;
cyl_home_fb_6   :BOOL;
cyl_work_fb_7   :BOOL;
cyl_home_fb_7   :BOOL;
cyl_work_fb_8   :BOOL;
cyl_home_fb_8   :BOOL;
cyl_work_fb_9   :BOOL;
cyl_home_fb_9   :BOOL;
cyl_work_fb_10  :BOOL;
cyl_home_fb_10  :BOOL;

// servo out

Actual_position_1       :real;
Actual_position_2       :real;
Actual_position_3       :real;
Actual_position_4       :real;
Actual_position_5       :real;
Actual_position_6       :real;
Actual_position_7       :real;
Actual_position_8       :real;
Actual_position_9       :real;
Actual_position_10      :real;

END_VAR
VAR_INPUT 
	
	//general
	offline_test      :BOOL;
	error_bit         :BOOL;
	
	// cylinder input set

cyl_work_sol_1        :BOOL;
cyl_home_sol_1        :BOOL;
delay_1_1             :LTIME;
delay_2_1             :LTIME;

cyl_work_sol_2        :BOOL;
cyl_home_sol_2        :BOOL;
delay_1_2             :LTIME;
delay_2_2             :LTIME;

cyl_work_sol_3        :BOOL;
cyl_home_sol_3        :BOOL;
delay_1_3             :LTIME;
delay_2_3             :LTIME;

cyl_work_sol_4        :BOOL;
cyl_home_sol_4        :BOOL;
delay_1_4             :LTIME;
delay_2_4             :LTIME;

cyl_work_sol_5        :BOOL;
cyl_home_sol_5        :BOOL;
delay_1_5             :LTIME;
delay_2_5             :LTIME;

cyl_work_sol_6        :BOOL;
cyl_home_sol_6        :BOOL;
delay_1_6             :LTIME;
delay_2_6             :LTIME;

cyl_work_sol_7        :BOOL;
cyl_home_sol_7        :BOOL;
delay_1_7             :LTIME;
delay_2_7             :LTIME;

cyl_work_sol_8        :BOOL;
cyl_home_sol_8        :BOOL;
delay_1_8             :LTIME;
delay_2_8             :LTIME;

cyl_work_sol_9        :BOOL;
cyl_home_sol_9        :BOOL;
delay_1_9             :LTIME;
delay_2_9             :LTIME;

cyl_work_sol_10       :bool;
cyl_home_sol_10       :BOOL;
delay_1_10            :LTIME;
delay_2_10            :LTIME;  
  
// servo input set

servo_absolute_1        :BOOL;
target_position_1       :REAL;
s_delay_1_1             :LTIME;

servo_absolute_2        :BOOL;
target_position_2       :REAL;
s_delay_1_2             :LTIME;

servo_absolute_3        :BOOL;
target_position_3       :REAL;
s_delay_1_3             :LTIME;

servo_absolute_4        :BOOL;
target_position_4       :REAL;
s_delay_1_4             :LTIME;

servo_absolute_5        :BOOL;
target_position_5       :REAL;
s_delay_1_5             :LTIME;

servo_absolute_6        :BOOL;
target_position_6       :REAL;
s_delay_1_6             :LTIME;

servo_absolute_7        :BOOL;
target_position_7       :REAL;
s_delay_1_7             :LTIME;

servo_absolute_8        :BOOL;
target_position_8       :REAL;
s_delay_1_8             :LTIME;

servo_absolute_9        :BOOL;
target_position_9       :REAL;
s_delay_1_9             :LTIME;

servo_absolute_10       :BOOL;
target_position_10      :REAL;
s_delay_1_10            :LTIME;

END_VAR

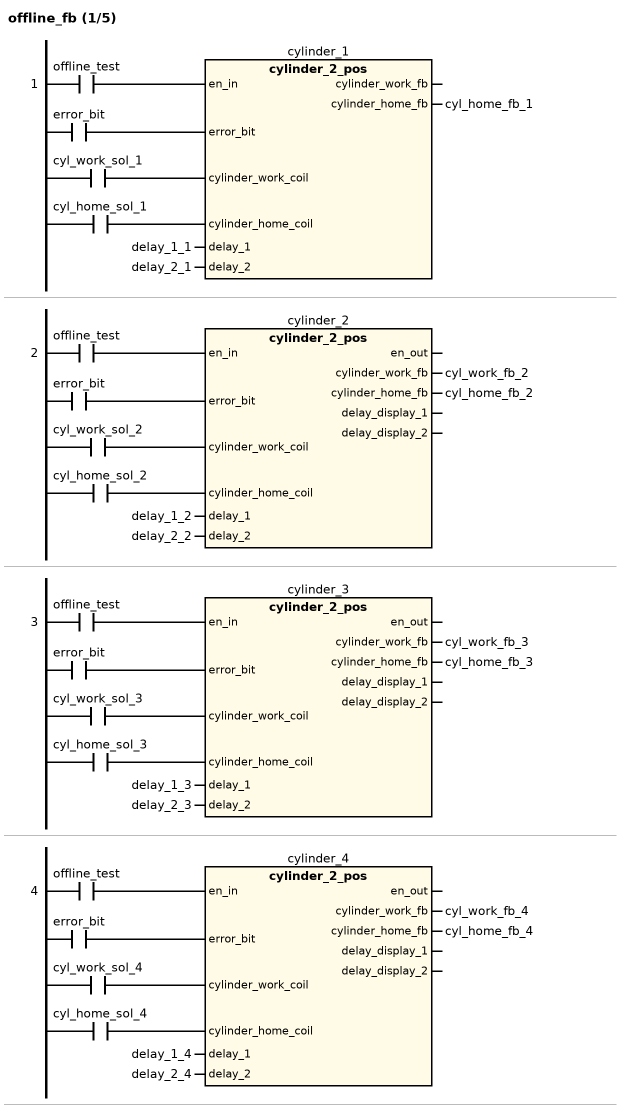
// NETWORK 1
cylinder_1(
    en_in := offline_test,
    error_bit := error_bit,
    cylinder_work_coil := cyl_work_sol_1,
    cylinder_home_coil := cyl_home_sol_1,
    delay_1 := delay_1_1,
    delay_2 := delay_2_1,
    cylinder_home_fb => cyl_home_fb_1); // cylinder_2_pos

// NETWORK 2
cylinder_2(
    en_in := offline_test,
    error_bit := error_bit,
    cylinder_work_coil := cyl_work_sol_2,
    cylinder_home_coil := cyl_home_sol_2,
    delay_1 := delay_1_2,
    delay_2 := delay_2_2,
    cylinder_work_fb => cyl_work_fb_2,
    cylinder_home_fb => cyl_home_fb_2); // cylinder_2_pos

// NETWORK 3
cylinder_3(
    en_in := offline_test,
    error_bit := error_bit,
    cylinder_work_coil := cyl_work_sol_3,
    cylinder_home_coil := cyl_home_sol_3,
    delay_1 := delay_1_3,
    delay_2 := delay_2_3,
    cylinder_work_fb => cyl_work_fb_3,
    cylinder_home_fb => cyl_home_fb_3); // cylinder_2_pos

// NETWORK 4
cylinder_4(
    en_in := offline_test,
    error_bit := error_bit,
    cylinder_work_coil := cyl_work_sol_4,
    cylinder_home_coil := cyl_home_sol_4,
    delay_1 := delay_1_4,
    delay_2 := delay_2_4,
    cylinder_work_fb => cyl_work_fb_4,
    cylinder_home_fb => cyl_home_fb_4); // cylinder_2_pos

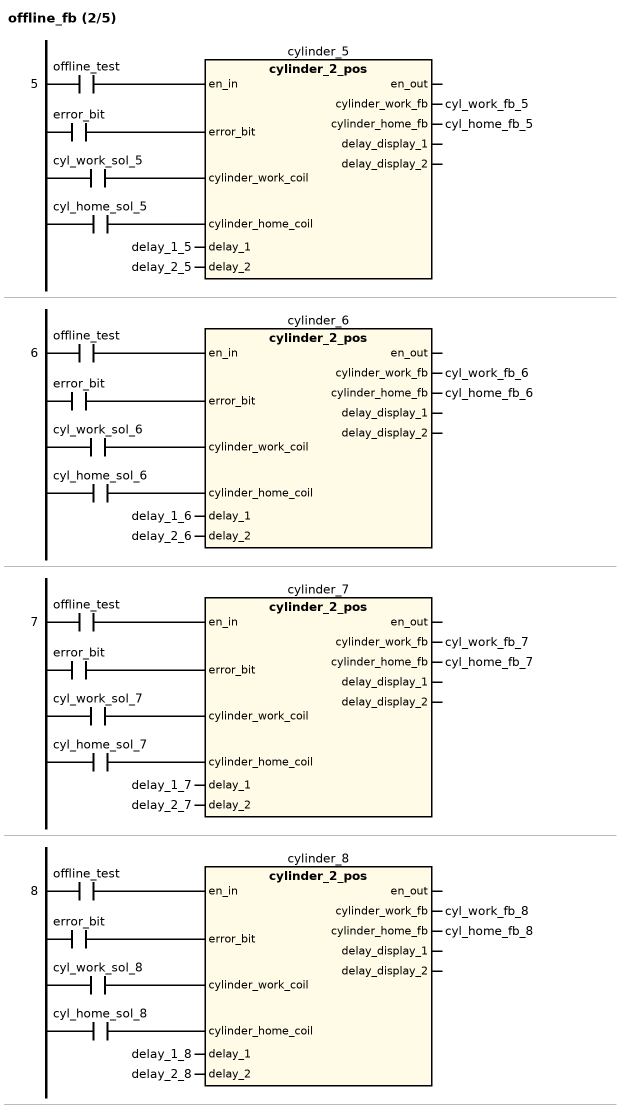
// NETWORK 5
cylinder_5(
    en_in := offline_test,
    error_bit := error_bit,
    cylinder_work_coil := cyl_work_sol_5,
    cylinder_home_coil := cyl_home_sol_5,
    delay_1 := delay_1_5,
    delay_2 := delay_2_5,
    cylinder_work_fb => cyl_work_fb_5,
    cylinder_home_fb => cyl_home_fb_5); // cylinder_2_pos

// NETWORK 6
cylinder_6(
    en_in := offline_test,
    error_bit := error_bit,
    cylinder_work_coil := cyl_work_sol_6,
    cylinder_home_coil := cyl_home_sol_6,
    delay_1 := delay_1_6,
    delay_2 := delay_2_6,
    cylinder_work_fb => cyl_work_fb_6,
    cylinder_home_fb => cyl_home_fb_6); // cylinder_2_pos

// NETWORK 7
cylinder_7(
    en_in := offline_test,
    error_bit := error_bit,
    cylinder_work_coil := cyl_work_sol_7,
    cylinder_home_coil := cyl_home_sol_7,
    delay_1 := delay_1_7,
    delay_2 := delay_2_7,
    cylinder_work_fb => cyl_work_fb_7,
    cylinder_home_fb => cyl_home_fb_7); // cylinder_2_pos

// NETWORK 8
cylinder_8(
    en_in := offline_test,
    error_bit := error_bit,
    cylinder_work_coil := cyl_work_sol_8,
    cylinder_home_coil := cyl_home_sol_8,
    delay_1 := delay_1_8,
    delay_2 := delay_2_8,
    cylinder_work_fb => cyl_work_fb_8,
    cylinder_home_fb => cyl_home_fb_8); // cylinder_2_pos

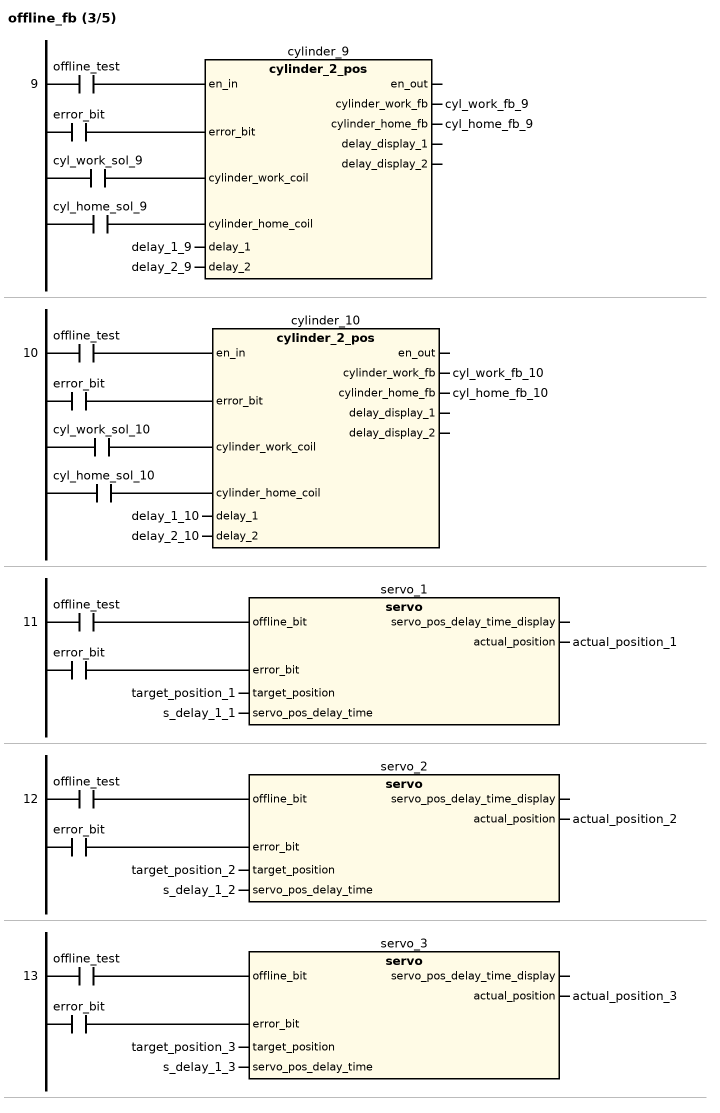
// NETWORK 9
cylinder_9(
    en_in := offline_test,
    error_bit := error_bit,
    cylinder_work_coil := cyl_work_sol_9,
    cylinder_home_coil := cyl_home_sol_9,
    delay_1 := delay_1_9,
    delay_2 := delay_2_9,
    cylinder_work_fb => cyl_work_fb_9,
    cylinder_home_fb => cyl_home_fb_9); // cylinder_2_pos

// NETWORK 10
cylinder_10(
    en_in := offline_test,
    error_bit := error_bit,
    cylinder_work_coil := cyl_work_sol_10,
    cylinder_home_coil := cyl_home_sol_10,
    delay_1 := delay_1_10,
    delay_2 := delay_2_10,
    cylinder_work_fb => cyl_work_fb_10,
    cylinder_home_fb => cyl_home_fb_10); // cylinder_2_pos

// NETWORK 11
servo_1(
    offline_bit := offline_test,
    error_bit := error_bit,
    target_position := target_position_1,
    servo_pos_delay_time := s_delay_1_1,
    actual_position => actual_position_1); // servo

// NETWORK 12
servo_2(
    offline_bit := offline_test,
    error_bit := error_bit,
    target_position := target_position_2,
    servo_pos_delay_time := s_delay_1_2,
    actual_position => actual_position_2); // servo

// NETWORK 13
servo_3(
    offline_bit := offline_test,
    error_bit := error_bit,
    target_position := target_position_3,
    servo_pos_delay_time := s_delay_1_3,
    actual_position => actual_position_3); // servo

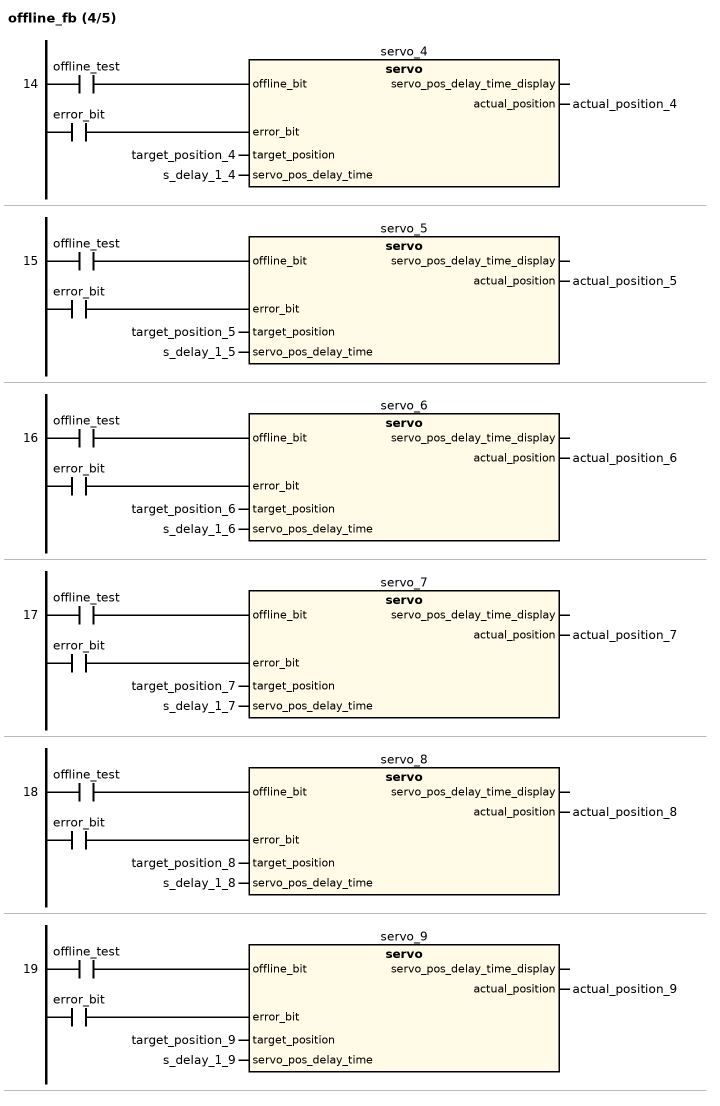
// NETWORK 14
servo_4(
    offline_bit := offline_test,
    error_bit := error_bit,
    target_position := target_position_4,
    servo_pos_delay_time := s_delay_1_4,
    actual_position => actual_position_4); // servo

// NETWORK 15
servo_5(
    offline_bit := offline_test,
    error_bit := error_bit,
    target_position := target_position_5,
    servo_pos_delay_time := s_delay_1_5,
    actual_position => actual_position_5); // servo

// NETWORK 16
servo_6(
    offline_bit := offline_test,
    error_bit := error_bit,
    target_position := target_position_6,
    servo_pos_delay_time := s_delay_1_6,
    actual_position => actual_position_6); // servo

// NETWORK 17
servo_7(
    offline_bit := offline_test,
    error_bit := error_bit,
    target_position := target_position_7,
    servo_pos_delay_time := s_delay_1_7,
    actual_position => actual_position_7); // servo

// NETWORK 18
servo_8(
    offline_bit := offline_test,
    error_bit := error_bit,
    target_position := target_position_8,
    servo_pos_delay_time := s_delay_1_8,
    actual_position => actual_position_8); // servo

// NETWORK 19
servo_9(
    offline_bit := offline_test,
    error_bit := error_bit,
    target_position := target_position_9,
    servo_pos_delay_time := s_delay_1_9,
    actual_position => actual_position_9); // servo

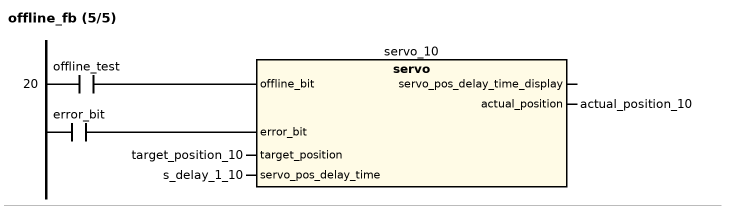
// NETWORK 20
servo_10(
    offline_bit := offline_test,
    error_bit := error_bit,
    target_position := target_position_10,
    servo_pos_delay_time := s_delay_1_10,
    actual_position => actual_position_10); // servo

END_FUNCTION_BLOCK

// ---- POUs/Programs/offline testing/offline_main.TcPOU
PROGRAM offline_main


VAR
	offline_1: offline_fb;
	offline_test: BOOL ;
	error_bit: BOOL;
	cyl_1_w_sol: BOOL;
	cyl_1_h_sol: BOOL;
	cyl_h_fb_1: BOOL;
	cyl_w_fb_1: BOOL;
END_VAR

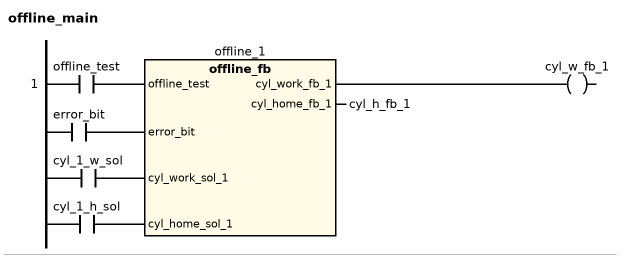
// NETWORK 1
offline_1(
    offline_test := offline_test,
    error_bit := error_bit,
    cyl_work_sol_1 := cyl_1_w_sol,
    cyl_home_sol_1 := cyl_1_h_sol,
    cyl_home_fb_1 => cyl_h_fb_1); // offline_fb
cyl_w_fb_1 := offline_1.cyl_work_fb_1;

END_PROGRAM

// ---- POUs/Programs/offline testing/POU_1.TcPOU
FUNCTION_BLOCK POU_1
VAR_INPUT
END_VAR
VAR_OUTPUT
END_VAR
VAR
END_VAR

// NETWORK 1

END_FUNCTION_BLOCK

// ---- POUs/Programs/offline testing/servo_validation.TcPOU
FUNCTION_BLOCK servo_validation

VAR_INPUT
offline_bit: BOOL;
error_bit: BOOL	;
servo_absolute: BOOL;
target_position: REAL;
servo_pos_delay_time: TIME;
END_VAR

VAR_OUTPUT
	servo_pos_delay_time_display: TIME;
	actual_position: REAL;
	absolute_done: BOOL;
END_VAR

VAR
	delay : ton;
END_VAR

// delay time move to timer
servo_pos_delay_time:=delay.PT;

// servo target position move to actual position
IF offline_bit AND NOT error_bit AND servo_absolute THEN
	delay.IN:=TRUE;
	IF delay.Q THEN
		absolute_done:=TRUE;
		actual_position:=target_position;
	END_IF
END_IF



// absolute done bit & timer in off
F_TRIG(CLK:=servo_absolute , Q=> );

IF f_trig.Q THEN
	absolute_done:=FALSE;
	delay.IN:=FALSE;
END_IF

END_FUNCTION_BLOCK

// ---- POUs/Programs/OP160/OP160_RFID.TcPOU
PROGRAM OP160_RFID
VAR
	OP160_RFID_TOOL: FB_RFID;
	OP160_RFID_FIX: FB_RFID;
	
	OP160_Tool_RFID_Read: BOOL;
	OP160_Tool_RFID_Write: BOOL;
	OP160_Tool_RFID_Quit: BOOL;
	OP160_HD_wrd_Num: INT;
	OP160_HD_wrd_Add: WORD;
END_VAR

OP160_RFID_TOOL(
	I_T_Timeout:= , 
	I_b_Head1SingleEnhanced:=TRUE , 
	I_b_Head1DataFixcode:= , 
	I_b_Head1SpecialFixcode:= , 
	I_b_Head1SpecialCommand:= , 
	I_b_Head1Read:=OP160_Tool_RFID_Read , 
	I_b_Head1Write:=OP160_Tool_RFID_Write , 
	I_b_Head1Quit:=OP160_Tool_RFID_Quit , 
	I_i_Head1WordNum:=OP160_HD_wrd_Num , 
	I_w_Head1WordAddress:=OP160_HD_wrd_Add , 
	I_w_Head1TagType:= , 
	HwIn:= , 
	IO_b_SetRestart:= , 
	IO_b_InitFinish:= , 
	Head1Data:= , 
	head1:= , 
	Memory:= , 
	O_b_Head1Busy=> , 
	O_b_Head1Done=> , 
	O_b_Head1NoDataCarrier=> , 
	O_b_Head1Error=> , 
	O_B_Head1Status=> , 
	O_B_Head1ReplyCounter=> , 
	HwOut=> );

END_PROGRAM
